LIN {X 0,Y 299.709,Z 498.448,A -85,B 0,C 180,E1 -16464.615,E2 -16464.615} C_VEL
LIN {X 0,Y 299.42,Z 499.838,A -85,B 0,C 180,E1 -16465.959,E2 -16465.959} C_VEL
LIN {X 0,Y 299.059,Z 501.418,A -85,B 0,C 180,E1 -16468.65,E2 -16468.65} C_VEL
LIN {X 0,Y 299.021,Z 501.647,A -85,B 0,C 180,E1 -16469.997,E2 -16469.997} C_VEL
LIN {X 0,Y 299.142,Z 500.888,A -85,B 0,C 180,E1 -16472.69,E2 -16472.69} C_VEL
LIN {X 0,Y 299.43,Z 499.927,A -85,B 0,C 180,E1 -16474.034,E2 -16474.034} C_VEL
LIN {X 0,Y 299.719,Z 498.589,A -85,B 0,C 180,E1 -16475.379,E2 -16475.379} C_VEL
LIN {X 0,Y 300.052,Z 495.813,A -85,B 0,C 180,E1 -16477.398,E2 -16477.398} C_VEL
LIN {X 0,Y 300.857,Z 491.982,A -85,B 0,C 180,E1 -16479.408,E2 -16479.408} C_VEL
LIN {X 0,Y 301.953,Z 486.999,A -85,B 0,C 180,E1 -16481.407,E2 -16481.407} C_VEL
LIN {X 0,Y 302.947,Z 480.761,A -85,B 0,C 180,E1 -16483.41,E2 -16483.41} C_VEL
LIN {X 0,Y 304.253,Z 472.973,A -85,B 0,C 180,E1 -16485.401,E2 -16485.401} C_VEL
LIN {X 0,Y 305.577,Z 464.983,A -85,B 0,C 180,E1 -16487.048,E2 -16487.048} C_VEL
LIN {X 0,Y 306.784,Z 456.263,A -85,B 0,C 180,E1 -16488.53,E2 -16488.53} C_VEL
LIN {X 0,Y 308.051,Z 445.435,A -85,B 0,C 180,E1 -16490.008,E2 -16490.008} C_VEL
LIN {X 0,Y 309.182,Z 435.113,A -85,B 0,C 180,E1 -16491.12,E2 -16491.12} C_VEL
LIN {X 0,Y 310.123,Z 422.899,A -85,B 0,C 180,E1 -16492.151,E2 -16492.151} C_VEL
LIN {X 0,Y 310.297,Z 416.875,A -85,B 0,C 180,E1 -16492.566,E2 -16492.566} C_VEL
LIN {X 0,Y 306.642,Z 404.751,A -85,B 0,C 180,E1 -16493.54,E2 -16493.54} C_VEL
LIN {X 0,Y 303.036,Z 394.815,A -85,B 0,C 180,E1 -16494.215,E2 -16494.215} C_VEL
LIN {X 0,Y 302.843,Z 385.653,A -85,B 0,C 180,E1 -16498.132,E2 -16498.132} C_VEL
LIN {X 0,Y 302.969,Z 376.735,A -85,B 0,C 180,E1 -16502.24,E2 -16502.24} C_VEL
LIN {X 0,Y 303.189,Z 369.244,A -85,B 0,C 180,E1 -16505.775,E2 -16505.775} C_VEL
LIN {X 0,Y 302.932,Z 365.032,A -85,B 0,C 180,E1 -16507.926,E2 -16507.926} C_VEL
LIN {X 0,Y 302.353,Z 361.246,A -85,B 0,C 180,E1 -16509.908,E2 -16509.908} C_VEL
LIN {X 0,Y 300.884,Z 354.027,A -85,B 0,C 180,E1 -16513.606,E2 -16513.606} C_VEL
LIN {X 0,Y 299.828,Z 349.15,A -85,B 0,C 180,E1 -16516.181,E2 -16516.181} C_VEL
LIN {X 0,Y 298.428,Z 343.625,A -85,B 0,C 180,E1 -16519.009,E2 -16519.009} C_VEL
LIN {X 0,Y 298.455,Z 343.623,A -85,B 0,C 180,E1 -16523.183,E2 -16523.183} C_VEL
LIN {X 0,Y 298.378,Z 343.625,A -85,B 0,C 180,E1 -16527.197,E2 -16527.197} C_VEL
LIN {X 0,Y 298.413,Z 343.62,A -85,B 0,C 180,E1 -16530.612,E2 -16530.612} C_VEL
LIN {X 0,Y 298.457,Z 343.611,A -85,B 0,C 180,E1 -16533.659,E2 -16533.659} C_VEL
LIN {X 0,Y 298.458,Z 343.612,A -85,B 0,C 180,E1 -16537.866,E2 -16537.866} C_VEL
LIN {X 0,Y 298.474,Z 343.618,A -85,B 0,C 180,E1 -16539.518,E2 -16539.518} C_VEL
LIN {X 0,Y 297.856,Z 343.69,A -85,B 0,C 180,E1 -16540.645,E2 -16540.645} C_VEL
LIN {X 0,Y 295.029,Z 344.044,A -85,B 0,C 180,E1 -16542.48,E2 -16542.48} C_VEL
LIN {X 0,Y 292.605,Z 344.349,A -85,B 0,C 180,E1 -16543.969,E2 -16543.969} C_VEL
LIN {X 0,Y 291.568,Z 344.467,A -85,B 0,C 180,E1 -16545.122,E2 -16545.122} C_VEL
LIN {X 0,Y 291.487,Z 344.474,A -85,B 0,C 180,E1 -16545.513,E2 -16545.513} C_VEL
LIN {X 0,Y 291.517,Z 344.482,A -85,B 0,C 180,E1 -16548.879,E2 -16548.879} C_VEL
LIN {X 0,Y 291.686,Z 344.456,A -85,B 0,C 180,E1 -16551.687,E2 -16551.687} C_VEL
LIN {X 0,Y 291.607,Z 344.465,A -85,B 0,C 180,E1 -16554.467,E2 -16554.467} C_VEL
LIN {X 0,Y 291.865,Z 344.442,A -85,B 0,C 180,E1 -16558.62,E2 -16558.62} C_VEL
LIN {X 0,Y 291.873,Z 344.427,A -85,B 0,C 180,E1 -16561.379,E2 -16561.379} C_VEL
LIN {X 0,Y 291.615,Z 344.473,A -85,B 0,C 180,E1 -16565.531,E2 -16565.531} C_VEL
LIN {X 0,Y 291.686,Z 344.464,A -85,B 0,C 180,E1 -16568.312,E2 -16568.312} C_VEL
LIN {X 0,Y 291.499,Z 344.489,A -85,B 0,C 180,E1 -16572.532,E2 -16572.532} C_VEL
LIN {X 0,Y 291.533,Z 344.484,A -85,B 0,C 180,E1 -16575.377,E2 -16575.377} C_VEL
LIN {X 0,Y 291.474,Z 344.489,A -85,B 0,C 180,E1 -16579.901,E2 -16579.901} C_VEL
LIN {X 0,Y 291.429,Z 344.53,A -85,B 0,C 180,E1 -16583.728,E2 -16583.728} C_VEL
LIN {X 0,Y 293.265,Z 351.385,A -85,B 0,C 180,E1 -16587.549,E2 -16587.549} C_VEL
LIN {X 0,Y 295.335,Z 359.255,A -85,B 0,C 180,E1 -16591.569,E2 -16591.569} C_VEL
LIN {X 0,Y 297.641,Z 367.228,A -85,B 0,C 180,E1 -16595.345,E2 -16595.345} C_VEL
LIN {X 0,Y 300.221,Z 376.648,A -85,B 0,C 180,E1 -16599.427,E2 -16599.427} C_VEL
LIN {X 0,Y 303.124,Z 387.143,A -85,B 0,C 180,E1 -16603.61,E2 -16603.61} C_VEL
LIN {X 0,Y 305.461,Z 395.462,A -85,B 0,C 180,E1 -16606.692,E2 -16606.692} C_VEL
LIN {X 0,Y 307.2,Z 402.134,A -85,B 0,C 180,E1 -16609.021,E2 -16609.021} C_VEL
LIN {X 0,Y 305.65,Z 408.163,A -85,B 0,C 180,E1 -16610.783,E2 -16610.783} C_VEL
LIN {X 0,Y 304.504,Z 412.249,A -85,B 0,C 180,E1 -16611.963,E2 -16611.963} C_VEL
LIN {X 0,Y 307.508,Z 435.324,A -85,B 0,C 180,E1 -16613.174,E2 -16613.174} C_VEL
LIN {X 0,Y 309.617,Z 451.923,A -85,B 0,C 180,E1 -16614.282,E2 -16614.282} C_VEL
LIN {X 0,Y 311.016,Z 467.45,A -85,B 0,C 180,E1 -16615.51,E2 -16615.51} C_VEL
LIN {X 0,Y 311.129,Z 472.166,A -85,B 0,C 180,E1 -16615.916,E2 -16615.916} C_VEL
LIN {X 0,Y 308.742,Z 487.07,A -85,B 0,C 180,E1 -16617.179,E2 -16617.179} C_VEL
LIN {X 0,Y 306.052,Z 501.73,A -85,B 0,C 180,E1 -16618.703,E2 -16618.703} C_VEL
LIN {X 0,Y 303.557,Z 514.784,A -85,B 0,C 180,E1 -16620.343,E2 -16620.343} C_VEL
LIN {X 0,Y 300.978,Z 527.029,A -85,B 0,C 180,E1 -16622.164,E2 -16622.164} C_VEL
LIN {X 0,Y 298.183,Z 540.238,A -85,B 0,C 180,E1 -16624.528,E2 -16624.528} C_VEL
LIN {X 0,Y 295.85,Z 551.36,A -85,B 0,C 180,E1 -16626.927,E2 -16626.927} C_VEL
LIN {X 0,Y 293.97,Z 560.802,A -85,B 0,C 180,E1 -16629.356,E2 -16629.356} C_VEL
LIN {X 0,Y 292.453,Z 569.92,A -85,B 0,C 180,E1 -16632.162,E2 -16632.162} C_VEL
LIN {X 0,Y 291.413,Z 576.815,A -85,B 0,C 180,E1 -16634.724,E2 -16634.724} C_VEL
LIN {X 0,Y 290.746,Z 582.794,A -85,B 0,C 180,E1 -16637.439,E2 -16637.439} C_VEL
LIN {X 0,Y 290.48,Z 587.668,A -85,B 0,C 180,E1 -16640.253,E2 -16640.253} C_VEL
LIN {X 0,Y 290.473,Z 591.326,A -85,B 0,C 180,E1 -16643.055,E2 -16643.055} C_VEL
LIN {X 0,Y 290.612,Z 593.786,A -85,B 0,C 180,E1 -16645.843,E2 -16645.843} C_VEL
LIN {X 0,Y 290.605,Z 595.006,A -85,B 0,C 180,E1 -16648.618,E2 -16648.618} C_VEL
LIN {X 0,Y 290.576,Z 595.145,A -85,B 0,C 180,E1 -16651.389,E2 -16651.389} C_VEL
LIN {X 0,Y 290.623,Z 594.104,A -85,B 0,C 180,E1 -16654.164,E2 -16654.164} C_VEL
LIN {X 0,Y 290.408,Z 591.736,A -85,B 0,C 180,E1 -16657.158,E2 -16657.158} C_VEL
LIN {X 0,Y 290.35,Z 588.681,A -85,B 0,C 180,E1 -16659.758,E2 -16659.758} C_VEL
LIN {X 0,Y 290.64,Z 584.298,A -85,B 0,C 180,E1 -16662.573,E2 -16662.573} C_VEL
LIN {X 0,Y 291.33,Z 578.847,A -85,B 0,C 180,E1 -16665.392,E2 -16665.392} C_VEL
LIN {X 0,Y 292.839,Z 570.307,A -85,B 0,C 180,E1 -16668.908,E2 -16668.908} C_VEL
LIN {X 0,Y 295.012,Z 560.871,A -85,B 0,C 180,E1 -16672.066,E2 -16672.066} C_VEL
LIN {X 0,Y 297.929,Z 549.828,A -85,B 0,C 180,E1 -16675.129,E2 -16675.129} C_VEL
LIN {X 0,Y 301.401,Z 538.282,A -85,B 0,C 180,E1 -16677.801,E2 -16677.801} C_VEL
LIN {X 0,Y 305.467,Z 524.903,A -85,B 0,C 180,E1 -16680.412,E2 -16680.412} C_VEL
LIN {X 0,Y 310.085,Z 510.339,A -85,B 0,C 180,E1 -16682.763,E2 -16682.763} C_VEL
LIN {X 0,Y 314.614,Z 495.802,A -85,B 0,C 180,E1 -16684.727,E2 -16684.727} C_VEL
LIN {X 0,Y 319.648,Z 479.136,A -85,B 0,C 180,E1 -16686.567,E2 -16686.567} C_VEL
LIN {X 0,Y 320.589,Z 474.856,A -85,B 0,C 180,E1 -16687.038,E2 -16687.038} C_VEL
LIN {X 0,Y 322.54,Z 461.569,A -85,B 0,C 180,E1 -16688.591,E2 -16688.591} C_VEL
LIN {X 0,Y 323.882,Z 451.061,A -85,B 0,C 180,E1 -16689.761,E2 -16689.761} C_VEL
LIN {X 0,Y 324.459,Z 439.447,A -85,B 0,C 180,E1 -16691.255,E2 -16691.255} C_VEL
LIN {X 0,Y 324.455,Z 428.956,A -85,B 0,C 180,E1 -16692.817,E2 -16692.817} C_VEL
LIN {X 0,Y 324.347,Z 427.026,A -85,B 0,C 180,E1 -16693.153,E2 -16693.153} C_VEL
LIN {X 0,Y 323.2,Z 424.156,A -85,B 0,C 180,E1 -16694.145,E2 -16694.145} C_VEL
LIN {X 0,Y 321.573,Z 421.326,A -85,B 0,C 180,E1 -16695.625,E2 -16695.625} C_VEL
LIN {X 0,Y 320.315,Z 419.287,A -85,B 0,C 180,E1 -16697.144,E2 -16697.144} C_VEL
LIN {X 0,Y 319.502,Z 417.856,A -85,B 0,C 180,E1 -16698.708,E2 -16698.708} C_VEL
LIN {X 0,Y 319.091,Z 417.219,A -85,B 0,C 180,E1 -16700.436,E2 -16700.436} C_VEL
LIN {X 0,Y 319.182,Z 417.312,A -85,B 0,C 180,E1 -16701.938,E2 -16701.938} C_VEL
LIN {X 0,Y 319.666,Z 420.051,A -85,B 0,C 180,E1 -16704.439,E2 -16704.439} C_VEL
LIN {X 0,Y 320.351,Z 423.999,A -85,B 0,C 180,E1 -16706.48,E2 -16706.48} C_VEL
LIN {X 0,Y 321.491,Z 428.847,A -85,B 0,C 180,E1 -16708.496,E2 -16708.496} C_VEL
LIN {X 0,Y 322.7,Z 435.191,A -85,B 0,C 180,E1 -16710.596,E2 -16710.596} C_VEL
LIN {X 0,Y 323.498,Z 442.422,A -85,B 0,C 180,E1 -16712.558,E2 -16712.558} C_VEL
LIN {X 0,Y 322.358,Z 446.313,A -85,B 0,C 180,E1 -16713.104,E2 -16713.104} C_VEL
LIN {X 0,Y 318.092,Z 458.146,A -85,B 0,C 180,E1 -16714.83,E2 -16714.83} C_VEL
LIN {X 0,Y 313.751,Z 469.712,A -85,B 0,C 180,E1 -16716.922,E2 -16716.922} C_VEL
LIN {X 0,Y 310.415,Z 478.194,A -85,B 0,C 180,E1 -16718.762,E2 -16718.762} C_VEL
LIN {X 0,Y 306.945,Z 486.567,A -85,B 0,C 180,E1 -16720.958,E2 -16720.958} C_VEL
LIN {X 0,Y 303.836,Z 493.445,A -85,B 0,C 180,E1 -16723.194,E2 -16723.194} C_VEL
LIN {X 0,Y 300.755,Z 499.656,A -85,B 0,C 180,E1 -16725.797,E2 -16725.797} C_VEL
LIN {X 0,Y 298.775,Z 503.283,A -85,B 0,C 180,E1 -16727.778,E2 -16727.778} C_VEL
LIN {X 0,Y 296.676,Z 506.657,A -85,B 0,C 180,E1 -16730.455,E2 -16730.455} C_VEL
LIN {X 0,Y 295.821,Z 507.785,A -85,B 0,C 180,E1 -16731.805,E2 -16731.805} C_VEL
LIN {X 0,Y 295.166,Z 508.504,A -85,B 0,C 180,E1 -16733.163,E2 -16733.163} C_VEL
LIN {X 0,Y 293.913,Z 508.817,A -85,B 0,C 180,E1 -16735.887,E2 -16735.887} C_VEL
LIN {X 0,Y 293.36,Z 508.405,A -85,B 0,C 180,E1 -16737.254,E2 -16737.254} C_VEL
LIN {X 0,Y 292.952,Z 507.587,A -85,B 0,C 180,E1 -16738.626,E2 -16738.626} C_VEL
LIN {X 0,Y 292.613,Z 506.375,A -85,B 0,C 180,E1 -16740.001,E2 -16740.001} C_VEL
LIN {X 0,Y 292.392,Z 503.757,A -85,B 0,C 180,E1 -16742.067,E2 -16742.067} C_VEL
LIN {X 0,Y 292.397,Z 500.192,A -85,B 0,C 180,E1 -16744.136,E2 -16744.136} C_VEL
LIN {X 0,Y 292.337,Z 495.653,A -85,B 0,C 180,E1 -16746.211,E2 -16746.211} C_VEL
LIN {X 0,Y 292.947,Z 488.932,A -85,B 0,C 180,E1 -16748.624,E2 -16748.624} C_VEL
LIN {X 0,Y 293.557,Z 480.592,A -85,B 0,C 180,E1 -16751.042,E2 -16751.042} C_VEL
LIN {X 0,Y 294.384,Z 471.876,A -85,B 0,C 180,E1 -16753.109,E2 -16753.109} C_VEL
LIN {X 0,Y 295.367,Z 461.466,A -85,B 0,C 180,E1 -16755.174,E2 -16755.174} C_VEL
LIN {X 0,Y 296.644,Z 450.12,A -85,B 0,C 180,E1 -16757.049,E2 -16757.049} C_VEL
LIN {X 0,Y 297.862,Z 437.703,A -85,B 0,C 180,E1 -16758.753,E2 -16758.753} C_VEL
LIN {X 0,Y 299.01,Z 424.062,A -85,B 0,C 180,E1 -16760.305,E2 -16760.305} C_VEL
LIN {X 0,Y 300.202,Z 410.631,A -85,B 0,C 180,E1 -16761.547,E2 -16761.547} C_VEL
LIN {X 0,Y 296.859,Z 394.61,A -85,B 0,C 180,E1 -16763.018,E2 -16763.018} C_VEL
LIN {X 0,Y 293.024,Z 378.623,A -85,B 0,C 180,E1 -16764.237,E2 -16764.237} C_VEL
LIN {X 0,Y 292.023,Z 374.499,A -85,B 0,C 180,E1 -16764.54,E2 -16764.54} C_VEL
LIN {X 0,Y 292.382,Z 369.177,A -85,B 0,C 180,E1 -16767.952,E2 -16767.952} C_VEL
LIN {X 0,Y 292.834,Z 363.258,A -85,B 0,C 180,E1 -16771.871,E2 -16771.871} C_VEL
LIN {X 0,Y 293.207,Z 358.041,A -85,B 0,C 180,E1 -16775.413,E2 -16775.413} C_VEL
LIN {X 0,Y 292.974,Z 353.615,A -85,B 0,C 180,E1 -16778.588,E2 -16778.588} C_VEL
LIN {X 0,Y 292.196,Z 348.783,A -85,B 0,C 180,E1 -16782.336,E2 -16782.336} C_VEL
LIN {X 0,Y 293.162,Z 351.814,A -85,B 0,C 180,E1 -16784.045,E2 -16784.045} C_VEL
LIN {X 0,Y 294.906,Z 359.618,A -85,B 0,C 180,E1 -16788.139,E2 -16788.139} C_VEL
LIN {X 0,Y 296.129,Z 366.652,A -85,B 0,C 180,E1 -16791.895,E2 -16791.895} C_VEL
LIN {X 0,Y 296.461,Z 370.31,A -85,B 0,C 180,E1 -16793.709,E2 -16793.709} C_VEL
LIN {X 0,Y 296.218,Z 378.746,A -85,B 0,C 180,E1 -16797.732,E2 -16797.732} C_VEL
LIN {X 0,Y 296.115,Z 389.045,A -85,B 0,C 180,E1 -16802.428,E2 -16802.428} C_VEL
LIN {X 0,Y 296.28,Z 395.804,A -85,B 0,C 180,E1 -16805.308,E2 -16805.308} C_VEL
LIN {X 0,Y 301.098,Z 409.41,A -85,B 0,C 180,E1 -16806.291,E2 -16806.291} C_VEL
LIN {X 0,Y 303.862,Z 419.007,A -85,B 0,C 180,E1 -16807.118,E2 -16807.118} C_VEL
LIN {X 0,Y 302.971,Z 431.867,A -85,B 0,C 180,E1 -16808.108,E2 -16808.108} C_VEL
LIN {X 0,Y 301.875,Z 443.495,A -85,B 0,C 180,E1 -16809.292,E2 -16809.292} C_VEL
LIN {X 0,Y 300.567,Z 454.315,A -85,B 0,C 180,E1 -16810.711,E2 -16810.711} C_VEL
LIN {X 0,Y 299.179,Z 463.594,A -85,B 0,C 180,E1 -16812.216,E2 -16812.216} C_VEL
LIN {X 0,Y 297.83,Z 472.044,A -85,B 0,C 180,E1 -16813.9,E2 -16813.9} C_VEL
LIN {X 0,Y 296.362,Z 480.26,A -85,B 0,C 180,E1 -16815.929,E2 -16815.929} C_VEL
LIN {X 0,Y 295.496,Z 485.81,A -85,B 0,C 180,E1 -16817.637,E2 -16817.637} C_VEL
LIN {X 0,Y 294.347,Z 491.24,A -85,B 0,C 180,E1 -16819.681,E2 -16819.681} C_VEL
LIN {X 0,Y 293.252,Z 495.521,A -85,B 0,C 180,E1 -16821.729,E2 -16821.729} C_VEL
LIN {X 0,Y 292.874,Z 497.74,A -85,B 0,C 180,E1 -16823.106,E2 -16823.106} C_VEL
LIN {X 0,Y 292.725,Z 499.525,A -85,B 0,C 180,E1 -16824.486,E2 -16824.486} C_VEL
LIN {X 0,Y 292.421,Z 500.915,A -85,B 0,C 180,E1 -16825.862,E2 -16825.862} C_VEL
LIN {X 0,Y 292.053,Z 502.493,A -85,B 0,C 180,E1 -16828.618,E2 -16828.618} C_VEL
LIN {X 0,Y 292.01,Z 502.723,A -85,B 0,C 180,E1 -16829.997,E2 -16829.997} C_VEL
LIN {X 0,Y 292.132,Z 501.964,A -85,B 0,C 180,E1 -16832.754,E2 -16832.754} C_VEL
LIN {X 0,Y 292.431,Z 501.003,A -85,B 0,C 180,E1 -16834.131,E2 -16834.131} C_VEL
LIN {X 0,Y 292.732,Z 499.664,A -85,B 0,C 180,E1 -16835.507,E2 -16835.507} C_VEL
LIN {X 0,Y 293.091,Z 496.889,A -85,B 0,C 180,E1 -16837.575,E2 -16837.575} C_VEL
LIN {X 0,Y 293.935,Z 493.056,A -85,B 0,C 180,E1 -16839.631,E2 -16839.631} C_VEL
LIN {X 0,Y 295.08,Z 488.072,A -85,B 0,C 180,E1 -16841.676,E2 -16841.676} C_VEL
LIN {X 0,Y 296.126,Z 481.832,A -85,B 0,C 180,E1 -16843.725,E2 -16843.725} C_VEL
LIN {X 0,Y 297.504,Z 474.04,A -85,B 0,C 180,E1 -16845.76,E2 -16845.76} C_VEL
LIN {X 0,Y 298.872,Z 466.05,A -85,B 0,C 180,E1 -16847.443,E2 -16847.443} C_VEL
LIN {X 0,Y 300.297,Z 456.215,A -85,B 0,C 180,E1 -16849.122,E2 -16849.122} C_VEL
LIN {X 0,Y 301.463,Z 446.492,A -85,B 0,C 180,E1 -16850.465,E2 -16850.465} C_VEL
LIN {X 0,Y 302.661,Z 436.146,A -85,B 0,C 180,E1 -16851.599,E2 -16851.599} C_VEL
LIN {X 0,Y 303.614,Z 424.465,A -85,B 0,C 180,E1 -16852.608,E2 -16852.608} C_VEL
LIN {X 0,Y 303.848,Z 418.707,A -85,B 0,C 180,E1 -16853.019,E2 -16853.019} C_VEL
LIN {X 0,Y 300.261,Z 406.801,A -85,B 0,C 180,E1 -16854.025,E2 -16854.025} C_VEL
LIN {X 0,Y 296.28,Z 395.811,A -85,B 0,C 180,E1 -16854.818,E2 -16854.818} C_VEL
LIN {X 0,Y 296.092,Z 387.112,A -85,B 0,C 180,E1 -16858.57,E2 -16858.57} C_VEL
LIN {X 0,Y 296.229,Z 379.14,A -85,B 0,C 180,E1 -16862.259,E2 -16862.259} C_VEL
LIN {X 0,Y 296.485,Z 370.58,A -85,B 0,C 180,E1 -16866.337,E2 -16866.337} C_VEL
LIN {X 0,Y 296.007,Z 365.472,A -85,B 0,C 180,E1 -16869.035,E2 -16869.035} C_VEL
LIN {X 0,Y 294.773,Z 359.052,A -85,B 0,C 180,E1 -16872.344,E2 -16872.344} C_VEL
LIN {X 0,Y 293.345,Z 352.213,A -85,B 0,C 180,E1 -16875.989,E2 -16875.989} C_VEL
LIN {X 0,Y 291.502,Z 345.062,A -85,B 0,C 180,E1 -16879.703,E2 -16879.703} C_VEL
LIN {X 0,Y 291.398,Z 344.498,A -85,B 0,C 180,E1 -16880.001,E2 -16880.001} C_VEL
LIN {X 0,Y 291.418,Z 344.499,A -85,B 0,C 180,E1 -16882.92,E2 -16882.92} C_VEL
LIN {X 0,Y 291.328,Z 344.506,A -85,B 0,C 180,E1 -16886.299,E2 -16886.299} C_VEL
LIN {X 0,Y 291.369,Z 344.496,A -85,B 0,C 180,E1 -16890.258,E2 -16890.258} C_VEL
LIN {X 0,Y 291.405,Z 344.492,A -85,B 0,C 180,E1 -16894.27,E2 -16894.27} C_VEL
LIN {X 0,Y 291.414,Z 344.487,A -85,B 0,C 180,E1 -16897.302,E2 -16897.302} C_VEL
LIN {X 0,Y 291.493,Z 344.483,A -85,B 0,C 180,E1 -16900.272,E2 -16900.272} C_VEL
LIN {X 0,Y 291.519,Z 344.477,A -85,B 0,C 180,E1 -16904.633,E2 -16904.633} C_VEL
LIN {X 0,Y 291.487,Z 344.474,A -85,B 0,C 180,E1 -16905.513,E2 -16905.513} C_VEL
LIN {X 0,Y 290.85,Z 344.559,A -85,B 0,C 180,E1 -16906.666,E2 -16906.666} C_VEL
LIN {X 0,Y 288.088,Z 344.912,A -85,B 0,C 180,E1 -16908.546,E2 -16908.546} C_VEL
LIN {X 0,Y 285.734,Z 345.2,A -85,B 0,C 180,E1 -16910.071,E2 -16910.071} C_VEL
LIN {X 0,Y 284.718,Z 345.322,A -85,B 0,C 180,E1 -16911.251,E2 -16911.251} C_VEL
LIN {X 0,Y 284.632,Z 345.333,A -85,B 0,C 180,E1 -16911.651,E2 -16911.651} C_VEL
LIN {X 0,Y 284.578,Z 345.342,A -85,B 0,C 180,E1 -16914.33,E2 -16914.33} C_VEL
LIN {X 0,Y 284.832,Z 345.318,A -85,B 0,C 180,E1 -16918.586,E2 -16918.586} C_VEL
LIN {X 0,Y 284.839,Z 345.303,A -85,B 0,C 180,E1 -16921.413,E2 -16921.413} C_VEL
LIN {X 0,Y 284.585,Z 345.35,A -85,B 0,C 180,E1 -16925.669,E2 -16925.669} C_VEL
LIN {X 0,Y 284.643,Z 345.341,A -85,B 0,C 180,E1 -16929.054,E2 -16929.054} C_VEL
LIN {X 0,Y 284.455,Z 345.365,A -85,B 0,C 180,E1 -16932.847,E2 -16932.847} C_VEL
LIN {X 0,Y 284.466,Z 345.365,A -85,B 0,C 180,E1 -16935.769,E2 -16935.769} C_VEL
LIN {X 0,Y 284.406,Z 345.369,A -85,B 0,C 180,E1 -16940.24,E2 -16940.24} C_VEL
LIN {X 0,Y 284.407,Z 345.509,A -85,B 0,C 180,E1 -16942.616,E2 -16942.616} C_VEL
LIN {X 0,Y 286.043,Z 351.774,A -85,B 0,C 180,E1 -16946.247,E2 -16946.247} C_VEL
LIN {X 0,Y 287.963,Z 358.811,A -85,B 0,C 180,E1 -16950.021,E2 -16950.021} C_VEL
LIN {X 0,Y 290.093,Z 366.587,A -85,B 0,C 180,E1 -16953.863,E2 -16953.863} C_VEL
LIN {X 0,Y 292.27,Z 374.529,A -85,B 0,C 180,E1 -16957.491,E2 -16957.491} C_VEL
LIN {X 0,Y 294.552,Z 382.807,A -85,B 0,C 180,E1 -16961.006,E2 -16961.006} C_VEL
LIN {X 0,Y 297.528,Z 393.255,A -85,B 0,C 180,E1 -16965.124,E2 -16965.124} C_VEL
LIN {X 0,Y 300.006,Z 402.705,A -85,B 0,C 180,E1 -16968.558,E2 -16968.558} C_VEL
LIN {X 0,Y 300.174,Z 404.143,A -85,B 0,C 180,E1 -16969.043,E2 -16969.043} C_VEL
LIN {X 0,Y 297.875,Z 412.008,A -85,B 0,C 180,E1 -16971.379,E2 -16971.379} C_VEL
LIN {X 0,Y 300.73,Z 434.611,A -85,B 0,C 180,E1 -16972.57,E2 -16972.57} C_VEL
LIN {X 0,Y 302.52,Z 449.258,A -85,B 0,C 180,E1 -16973.548,E2 -16973.548} C_VEL
LIN {X 0,Y 304.076,Z 465.037,A -85,B 0,C 180,E1 -16974.816,E2 -16974.816} C_VEL
LIN {X 0,Y 304.479,Z 472.307,A -85,B 0,C 180,E1 -16975.467,E2 -16975.467} C_VEL
LIN {X 0,Y 301.82,Z 488.204,A -85,B 0,C 180,E1 -16976.868,E2 -16976.868} C_VEL
LIN {X 0,Y 299.001,Z 502.917,A -85,B 0,C 180,E1 -16978.472,E2 -16978.472} C_VEL
LIN {X 0,Y 296.435,Z 515.616,A -85,B 0,C 180,E1 -16980.145,E2 -16980.145} C_VEL
LIN {X 0,Y 293.704,Z 528.288,A -85,B 0,C 180,E1 -16982.128,E2 -16982.128} C_VEL
LIN {X 0,Y 291.234,Z 539.758,A -85,B 0,C 180,E1 -16984.259,E2 -16984.259} C_VEL
LIN {X 0,Y 288.848,Z 550.829,A -85,B 0,C 180,E1 -16986.715,E2 -16986.715} C_VEL
LIN {X 0,Y 286.954,Z 560.211,A -85,B 0,C 180,E1 -16989.203,E2 -16989.203} C_VEL
LIN {X 0,Y 285.395,Z 569.257,A -85,B 0,C 180,E1 -16992.076,E2 -16992.076} C_VEL
LIN {X 0,Y 284.231,Z 576.989,A -85,B 0,C 180,E1 -16995.096,E2 -16995.096} C_VEL
LIN {X 0,Y 283.672,Z 582.686,A -85,B 0,C 180,E1 -16997.847,E2 -16997.847} C_VEL
LIN {X 0,Y 283.434,Z 587.361,A -85,B 0,C 180,E1 -17000.729,E2 -17000.729} C_VEL
LIN {X 0,Y 283.479,Z 590.049,A -85,B 0,C 180,E1 -17002.883,E2 -17002.883} C_VEL
LIN {X 0,Y 283.587,Z 592.542,A -85,B 0,C 180,E1 -17005.74,E2 -17005.74} C_VEL
LIN {X 0,Y 283.596,Z 593.839,A -85,B 0,C 180,E1 -17008.583,E2 -17008.583} C_VEL
LIN {X 0,Y 283.56,Z 594.03,A -85,B 0,C 180,E1 -17011.424,E2 -17011.424} C_VEL
LIN {X 0,Y 283.591,Z 593.024,A -85,B 0,C 180,E1 -17014.267,E2 -17014.267} C_VEL
LIN {X 0,Y 283.351,Z 590.857,A -85,B 0,C 180,E1 -17017.2,E2 -17017.2} C_VEL
LIN {X 0,Y 283.28,Z 587.686,A -85,B 0,C 180,E1 -17020.004,E2 -17020.004} C_VEL
LIN {X 0,Y 283.603,Z 583.386,A -85,B 0,C 180,E1 -17022.89,E2 -17022.89} C_VEL
LIN {X 0,Y 284.342,Z 577.983,A -85,B 0,C 180,E1 -17025.78,E2 -17025.78} C_VEL
LIN {X 0,Y 285.569,Z 571.386,A -85,B 0,C 180,E1 -17028.662,E2 -17028.662} C_VEL
LIN {X 0,Y 287.581,Z 562.85,A -85,B 0,C 180,E1 -17031.775,E2 -17031.775} C_VEL
LIN {X 0,Y 290.234,Z 553.302,A -85,B 0,C 180,E1 -17034.693,E2 -17034.693} C_VEL
LIN {X 0,Y 293.823,Z 541.818,A -85,B 0,C 180,E1 -17037.629,E2 -17037.629} C_VEL
LIN {X 0,Y 297.617,Z 530.286,A -85,B 0,C 180,E1 -17040.122,E2 -17040.122} C_VEL
LIN {X 0,Y 302.489,Z 516.005,A -85,B 0,C 180,E1 -17042.699,E2 -17042.699} C_VEL
LIN {X 0,Y 307.398,Z 501.59,A -85,B 0,C 180,E1 -17044.863,E2 -17044.863} C_VEL
LIN {X 0,Y 312.17,Z 487.424,A -85,B 0,C 180,E1 -17046.63,E2 -17046.63} C_VEL
LIN {X 0,Y 315.197,Z 477.495,A -85,B 0,C 180,E1 -17047.725,E2 -17047.725} C_VEL
LIN {X 0,Y 317.501,Z 464.627,A -85,B 0,C 180,E1 -17049.327,E2 -17049.327} C_VEL
LIN {X 0,Y 319.351,Z 453.739,A -85,B 0,C 180,E1 -17050.607,E2 -17050.607} C_VEL
LIN {X 0,Y 320.344,Z 442.456,A -85,B 0,C 180,E1 -17052.137,E2 -17052.137} C_VEL
LIN {X 0,Y 320.788,Z 432.6,A -85,B 0,C 180,E1 -17053.699,E2 -17053.699} C_VEL
LIN {X 0,Y 319.912,Z 429.825,A -85,B 0,C 180,E1 -17054.671,E2 -17054.671} C_VEL
LIN {X 0,Y 317.988,Z 426.453,A -85,B 0,C 180,E1 -17056.754,E2 -17056.754} C_VEL
LIN {X 0,Y 316.786,Z 424.341,A -85,B 0,C 180,E1 -17058.968,E2 -17058.968} C_VEL
LIN {X 0,Y 316.365,Z 423.813,A -85,B 0,C 180,E1 -17061.537,E2 -17061.537} C_VEL
LIN {X 0,Y 316.5,Z 426.109,A -85,B 0,C 180,E1 -17064.028,E2 -17064.028} C_VEL
LIN {X 0,Y 316.78,Z 428.779,A -85,B 0,C 180,E1 -17065.626,E2 -17065.626} C_VEL
LIN {X 0,Y 317.486,Z 433.861,A -85,B 0,C 180,E1 -17067.909,E2 -17067.909} C_VEL
LIN {X 0,Y 318.083,Z 438.239,A -85,B 0,C 180,E1 -17069.512,E2 -17069.512} C_VEL
LIN {X 0,Y 318.614,Z 444.125,A -85,B 0,C 180,E1 -17071.326,E2 -17071.326} C_VEL
LIN {X 0,Y 318.599,Z 446.482,A -85,B 0,C 180,E1 -17071.933,E2 -17071.933} C_VEL
LIN {X 0,Y 313.832,Z 458.914,A -85,B 0,C 180,E1 -17073.751,E2 -17073.751} C_VEL
LIN {X 0,Y 309.106,Z 470.425,A -85,B 0,C 180,E1 -17075.842,E2 -17075.842} C_VEL
LIN {X 0,Y 305.061,Z 479.771,A -85,B 0,C 180,E1 -17077.914,E2 -17077.914} C_VEL
LIN {X 0,Y 301.2,Z 488.323,A -85,B 0,C 180,E1 -17080.225,E2 -17080.225} C_VEL
LIN {X 0,Y 298.329,Z 494.204,A -85,B 0,C 180,E1 -17082.167,E2 -17082.167} C_VEL
LIN {X 0,Y 295.005,Z 500.52,A -85,B 0,C 180,E1 -17084.808,E2 -17084.808} C_VEL
LIN {X 0,Y 292.115,Z 505.237,A -85,B 0,C 180,E1 -17087.495,E2 -17087.495} C_VEL
LIN {X 0,Y 289.908,Z 508.421,A -85,B 0,C 180,E1 -17090.23,E2 -17090.23} C_VEL
LIN {X 0,Y 288.287,Z 510.026,A -85,B 0,C 180,E1 -17092.999,E2 -17092.999} C_VEL
LIN {X 0,Y 286.961,Z 510.141,A -85,B 0,C 180,E1 -17095.787,E2 -17095.787} C_VEL
LIN {X 0,Y 285.951,Z 508.743,A -85,B 0,C 180,E1 -17098.592,E2 -17098.592} C_VEL
LIN {X 0,Y 285.599,Z 507.45,A -85,B 0,C 180,E1 -17100.001,E2 -17100.001} C_VEL
LIN {X 0,Y 285.36,Z 504.691,A -85,B 0,C 180,E1 -17102.118,E2 -17102.118} C_VEL
LIN {X 0,Y 285.382,Z 500.98,A -85,B 0,C 180,E1 -17104.237,E2 -17104.237} C_VEL
LIN {X 0,Y 285.323,Z 496.3,A -85,B 0,C 180,E1 -17106.364,E2 -17106.364} C_VEL
LIN {X 0,Y 285.961,Z 489.426,A -85,B 0,C 180,E1 -17108.836,E2 -17108.836} C_VEL
LIN {X 0,Y 286.6,Z 480.915,A -85,B 0,C 180,E1 -17111.314,E2 -17111.314} C_VEL
LIN {X 0,Y 287.438,Z 472.012,A -85,B 0,C 180,E1 -17113.432,E2 -17113.432} C_VEL
LIN {X 0,Y 288.465,Z 461.403,A -85,B 0,C 180,E1 -17115.546,E2 -17115.546} C_VEL
LIN {X 0,Y 289.825,Z 449.814,A -85,B 0,C 180,E1 -17117.463,E2 -17117.463} C_VEL
LIN {X 0,Y 291.216,Z 435.81,A -85,B 0,C 180,E1 -17119.381,E2 -17119.381} C_VEL
LIN {X 0,Y 292.448,Z 422.003,A -85,B 0,C 180,E1 -17120.927,E2 -17120.927} C_VEL
LIN {X 0,Y 293.347,Z 411.729,A -85,B 0,C 180,E1 -17121.889,E2 -17121.889} C_VEL
LIN {X 0,Y 290.216,Z 396.576,A -85,B 0,C 180,E1 -17123.325,E2 -17123.325} C_VEL
LIN {X 0,Y 286.689,Z 381.561,A -85,B 0,C 180,E1 -17124.529,E2 -17124.529} C_VEL
LIN {X 0,Y 285.049,Z 374.919,A -85,B 0,C 180,E1 -17125.025,E2 -17125.025} C_VEL
LIN {X 0,Y 285.587,Z 368.101,A -85,B 0,C 180,E1 -17129.485,E2 -17129.485} C_VEL
LIN {X 0,Y 286.011,Z 362.421,A -85,B 0,C 180,E1 -17133.332,E2 -17133.332} C_VEL
LIN {X 0,Y 286.196,Z 358.446,A -85,B 0,C 180,E1 -17136.112,E2 -17136.112} C_VEL
LIN {X 0,Y 285.958,Z 354.675,A -85,B 0,C 180,E1 -17138.873,E2 -17138.873} C_VEL
LIN {X 0,Y 285.335,Z 350.833,A -85,B 0,C 180,E1 -17141.92,E2 -17141.92} C_VEL
LIN {X 0,Y 286.647,Z 354.638,A -85,B 0,C 180,E1 -17144.064,E2 -17144.064} C_VEL
LIN {X 0,Y 288.225,Z 361.926,A -85,B 0,C 180,E1 -17147.981,E2 -17147.981} C_VEL
LIN {X 0,Y 289.266,Z 367.635,A -85,B 0,C 180,E1 -17151.03,E2 -17151.03} C_VEL
LIN {X 0,Y 289.74,Z 371.784,A -85,B 0,C 180,E1 -17153.175,E2 -17153.175} C_VEL
LIN {X 0,Y 289.539,Z 379.493,A -85,B 0,C 180,E1 -17156.894,E2 -17156.894} C_VEL
LIN {X 0,Y 289.363,Z 388.266,A -85,B 0,C 180,E1 -17160.971,E2 -17160.971} C_VEL
LIN {X 0,Y 289.529,Z 396.869,A -85,B 0,C 180,E1 -17164.711,E2 -17164.711} C_VEL
LIN {X 0,Y 294.179,Z 409.674,A -85,B 0,C 180,E1 -17165.652,E2 -17165.652} C_VEL
LIN {X 0,Y 297.311,Z 420.264,A -85,B 0,C 180,E1 -17166.599,E2 -17166.599} C_VEL
LIN {X 0,Y 296.498,Z 432.72,A -85,B 0,C 180,E1 -17167.584,E2 -17167.584} C_VEL
LIN {X 0,Y 295.324,Z 444.516,A -85,B 0,C 180,E1 -17168.805,E2 -17168.805} C_VEL
LIN {X 0,Y 293.95,Z 455.384,A -85,B 0,C 180,E1 -17170.259,E2 -17170.259} C_VEL
LIN {X 0,Y 292.519,Z 464.663,A -85,B 0,C 180,E1 -17171.797,E2 -17171.797} C_VEL
LIN {X 0,Y 291.095,Z 473.118,A -85,B 0,C 180,E1 -17173.517,E2 -17173.517} C_VEL
LIN {X 0,Y 289.561,Z 481.336,A -85,B 0,C 180,E1 -17175.591,E2 -17175.591} C_VEL
LIN {X 0,Y 288.652,Z 486.885,A -85,B 0,C 180,E1 -17177.339,E2 -17177.339} C_VEL
LIN {X 0,Y 287.446,Z 492.316,A -85,B 0,C 180,E1 -17179.43,E2 -17179.43} C_VEL
LIN {X 0,Y 286.31,Z 496.598,A -85,B 0,C 180,E1 -17181.527,E2 -17181.527} C_VEL
LIN {X 0,Y 285.909,Z 498.817,A -85,B 0,C 180,E1 -17182.937,E2 -17182.937} C_VEL
LIN {X 0,Y 285.74,Z 500.602,A -85,B 0,C 180,E1 -17184.351,E2 -17184.351} C_VEL
LIN {X 0,Y 285.422,Z 501.992,A -85,B 0,C 180,E1 -17185.76,E2 -17185.76} C_VEL
LIN {X 0,Y 285.044,Z 503.569,A -85,B 0,C 180,E1 -17188.584,E2 -17188.584} C_VEL
LIN {X 0,Y 285.019,Z 503.796,A -85,B 0,C 180,E1 -17189.997,E2 -17189.997} C_VEL
LIN {X 0,Y 285.124,Z 503.041,A -85,B 0,C 180,E1 -17192.822,E2 -17192.822} C_VEL
LIN {X 0,Y 285.432,Z 502.079,A -85,B 0,C 180,E1 -17194.233,E2 -17194.233} C_VEL
LIN {X 0,Y 285.746,Z 500.741,A -85,B 0,C 180,E1 -17195.642,E2 -17195.642} C_VEL
LIN {X 0,Y 286.133,Z 497.964,A -85,B 0,C 180,E1 -17197.76,E2 -17197.76} C_VEL
LIN {X 0,Y 287.019,Z 494.131,A -85,B 0,C 180,E1 -17199.866,E2 -17199.866} C_VEL
LIN {X 0,Y 288.213,Z 489.145,A -85,B 0,C 180,E1 -17201.959,E2 -17201.959} C_VEL
LIN {X 0,Y 289.312,Z 482.904,A -85,B 0,C 180,E1 -17204.055,E2 -17204.055} C_VEL
LIN {X 0,Y 290.775,Z 475.107,A -85,B 0,C 180,E1 -17206.134,E2 -17206.134} C_VEL
LIN {X 0,Y 292.182,Z 467.116,A -85,B 0,C 180,E1 -17207.855,E2 -17207.855} C_VEL
LIN {X 0,Y 293.678,Z 457.277,A -85,B 0,C 180,E1 -17209.571,E2 -17209.571} C_VEL
LIN {X 0,Y 294.894,Z 447.55,A -85,B 0,C 180,E1 -17210.942,E2 -17210.942} C_VEL
LIN {X 0,Y 296.149,Z 437.135,A -85,B 0,C 180,E1 -17212.106,E2 -17212.106} C_VEL
LIN {X 0,Y 297.113,Z 425.787,A -85,B 0,C 180,E1 -17213.107,E2 -17213.107} C_VEL
LIN {X 0,Y 297.414,Z 421.198,A -85,B 0,C 180,E1 -17213.437,E2 -17213.437} C_VEL
LIN {X 0,Y 294.605,Z 410.997,A -85,B 0,C 180,E1 -17214.351,E2 -17214.351} C_VEL
LIN {X 0,Y 290.422,Z 399.211,A -85,B 0,C 180,E1 -17215.251,E2 -17215.251} C_VEL
LIN {X 0,Y 289.506,Z 396.85,A -85,B 0,C 180,E1 -17215.44,E2 -17215.44} C_VEL
LIN {X 0,Y 289.388,Z 388.515,A -85,B 0,C 180,E1 -17219.055,E2 -17219.055} C_VEL
LIN {X 0,Y 289.571,Z 379.831,A -85,B 0,C 180,E1 -17223.094,E2 -17223.094} C_VEL
LIN {X 0,Y 289.822,Z 373.437,A -85,B 0,C 180,E1 -17226.2,E2 -17226.2} C_VEL
LIN {X 0,Y 289.541,Z 369.543,A -85,B 0,C 180,E1 -17228.154,E2 -17228.154} C_VEL
LIN {X 0,Y 288.637,Z 364.019,A -85,B 0,C 180,E1 -17231.098,E2 -17231.098} C_VEL
LIN {X 0,Y 287.114,Z 356.389,A -85,B 0,C 180,E1 -17235.218,E2 -17235.218} C_VEL
LIN {X 0,Y 285.635,Z 350.337,A -85,B 0,C 180,E1 -17238.368,E2 -17238.368} C_VEL
LIN {X 0,Y 284.328,Z 345.379,A -85,B 0,C 180,E1 -17241.154,E2 -17241.154} C_VEL
LIN {X 0,Y 284.346,Z 345.374,A -85,B 0,C 180,E1 -17244.643,E2 -17244.643} C_VEL
LIN {X 0,Y 284.278,Z 345.389,A -85,B 0,C 180,E1 -17248.723,E2 -17248.723} C_VEL
LIN {X 0,Y 284.379,Z 345.367,A -85,B 0,C 180,E1 -17252.824,E2 -17252.824} C_VEL
LIN {X 0,Y 284.376,Z 345.365,A -85,B 0,C 180,E1 -17256.707,E2 -17256.707} C_VEL
LIN {X 0,Y 284.416,Z 345.367,A -85,B 0,C 180,E1 -17259.869,E2 -17259.869} C_VEL
LIN {X 0,Y 284.457,Z 345.359,A -85,B 0,C 180,E1 -17264.468,E2 -17264.468} C_VEL
LIN {X 0,Y 284.469,Z 345.362,A -85,B 0,C 180,E1 -17268.6,E2 -17268.6} C_VEL
LIN {X 0,Y 284.632,Z 345.333,A -85,B 0,C 180,E1 -17271.651,E2 -17271.651} C_VEL
LIN {X 0,Y 283.951,Z 345.429,A -85,B 0,C 180,E1 -17272.83,E2 -17272.83} C_VEL
LIN {X 0,Y 281.096,Z 345.774,A -85,B 0,C 180,E1 -17274.752,E2 -17274.752} C_VEL
LIN {X 0,Y 278.725,Z 346.069,A -85,B 0,C 180,E1 -17276.313,E2 -17276.313} C_VEL
LIN {X 0,Y 277.769,Z 346.197,A -85,B 0,C 180,E1 -17277.523,E2 -17277.523} C_VEL
LIN {X 0,Y 277.723,Z 346.199,A -85,B 0,C 180,E1 -17277.932,E2 -17277.932} C_VEL
LIN {X 0,Y 277.849,Z 346.174,A -85,B 0,C 180,E1 -17279.999,E2 -17279.999} C_VEL
LIN {X 0,Y 277.695,Z 346.208,A -85,B 0,C 180,E1 -17282.901,E2 -17282.901} C_VEL
LIN {X 0,Y 277.632,Z 346.214,A -85,B 0,C 180,E1 -17287.271,E2 -17287.271} C_VEL
LIN {X 0,Y 277.485,Z 346.235,A -85,B 0,C 180,E1 -17290.212,E2 -17290.212} C_VEL
LIN {X 0,Y 277.413,Z 346.242,A -85,B 0,C 180,E1 -17294.675,E2 -17294.675} C_VEL
LIN {X 0,Y 277.355,Z 346.25,A -85,B 0,C 180,E1 -17299.232,E2 -17299.232} C_VEL
LIN {X 0,Y 277.327,Z 346.305,A -85,B 0,C 180,E1 -17301.363,E2 -17301.363} C_VEL
LIN {X 0,Y 279.116,Z 352.899,A -85,B 0,C 180,E1 -17305.343,E2 -17305.343} C_VEL
LIN {X 0,Y 280.969,Z 359.861,A -85,B 0,C 180,E1 -17309.192,E2 -17309.192} C_VEL
LIN {X 0,Y 283.491,Z 369.18,A -85,B 0,C 180,E1 -17313.903,E2 -17313.903} C_VEL
LIN {X 0,Y 285.351,Z 376.076,A -85,B 0,C 180,E1 -17317.114,E2 -17317.114} C_VEL
LIN {X 0,Y 287.661,Z 384.486,A -85,B 0,C 180,E1 -17320.773,E2 -17320.773} C_VEL
LIN {X 0,Y 290.7,Z 395.119,A -85,B 0,C 180,E1 -17325.064,E2 -17325.064} C_VEL
LIN {X 0,Y 293.226,Z 405.19,A -85,B 0,C 180,E1 -17328.773,E2 -17328.773} C_VEL
LIN {X 0,Y 291.36,Z 411.512,A -85,B 0,C 180,E1 -17330.72,E2 -17330.72} C_VEL
LIN {X 0,Y 294.186,Z 435.721,A -85,B 0,C 180,E1 -17332.069,E2 -17332.069} C_VEL
LIN {X 0,Y 296.135,Z 452.388,A -85,B 0,C 180,E1 -17333.262,E2 -17333.262} C_VEL
LIN {X 0,Y 297.556,Z 468.646,A -85,B 0,C 180,E1 -17334.654,E2 -17334.654} C_VEL
LIN {X 0,Y 297.651,Z 473.35,A -85,B 0,C 180,E1 -17335.077,E2 -17335.077} C_VEL
LIN {X 0,Y 294.909,Z 489.006,A -85,B 0,C 180,E1 -17336.52,E2 -17336.52} C_VEL
LIN {X 0,Y 291.961,Z 503.996,A -85,B 0,C 180,E1 -17338.231,E2 -17338.231} C_VEL
LIN {X 0,Y 289.341,Z 516.363,A -85,B 0,C 180,E1 -17339.94,E2 -17339.94} C_VEL
LIN {X 0,Y 286.623,Z 528.766,A -85,B 0,C 180,E1 -17341.971,E2 -17341.971} C_VEL
LIN {X 0,Y 283.93,Z 540.86,A -85,B 0,C 180,E1 -17344.336,E2 -17344.336} C_VEL
LIN {X 0,Y 281.54,Z 551.773,A -85,B 0,C 180,E1 -17346.892,E2 -17346.892} C_VEL
LIN {X 0,Y 279.696,Z 560.81,A -85,B 0,C 180,E1 -17349.408,E2 -17349.408} C_VEL
LIN {X 0,Y 278.2,Z 569.575,A -85,B 0,C 180,E1 -17352.357,E2 -17352.357} C_VEL
LIN {X 0,Y 277.128,Z 576.719,A -85,B 0,C 180,E1 -17355.313,E2 -17355.313} C_VEL
LIN {X 0,Y 276.568,Z 582.471,A -85,B 0,C 180,E1 -17358.274,E2 -17358.274} C_VEL
LIN {X 0,Y 276.4,Z 586.947,A -85,B 0,C 180,E1 -17361.228,E2 -17361.228} C_VEL
LIN {X 0,Y 276.458,Z 588.727,A -85,B 0,C 180,E1 -17362.701,E2 -17362.701} C_VEL
LIN {X 0,Y 276.565,Z 591.274,A -85,B 0,C 180,E1 -17365.631,E2 -17365.631} C_VEL
LIN {X 0,Y 276.59,Z 592.658,A -85,B 0,C 180,E1 -17368.548,E2 -17368.548} C_VEL
LIN {X 0,Y 276.596,Z 592.937,A -85,B 0,C 180,E1 -17370.004,E2 -17370.004} C_VEL
LIN {X 0,Y 276.531,Z 592.538,A -85,B 0,C 180,E1 -17372.917,E2 -17372.917} C_VEL
LIN {X 0,Y 276.559,Z 591.942,A -85,B 0,C 180,E1 -17374.376,E2 -17374.376} C_VEL
LIN {X 0,Y 276.291,Z 589.903,A -85,B 0,C 180,E1 -17377.31,E2 -17377.31} C_VEL
LIN {X 0,Y 276.236,Z 586.701,A -85,B 0,C 180,E1 -17380.262,E2 -17380.262} C_VEL
LIN {X 0,Y 276.584,Z 582.496,A -85,B 0,C 180,E1 -17383.223,E2 -17383.223} C_VEL
LIN {X 0,Y 277.356,Z 577.14,A -85,B 0,C 180,E1 -17386.188,E2 -17386.188} C_VEL
LIN {X 0,Y 278.693,Z 570.674,A -85,B 0,C 180,E1 -17389.14,E2 -17389.14} C_VEL
LIN {X 0,Y 280.692,Z 562.923,A -85,B 0,C 180,E1 -17392.12,E2 -17392.12} C_VEL
LIN {X 0,Y 283.657,Z 552.967,A -85,B 0,C 180,E1 -17395.305,E2 -17395.305} C_VEL
LIN {X 0,Y 287.707,Z 541.177,A -85,B 0,C 180,E1 -17398.432,E2 -17398.432} C_VEL
LIN {X 0,Y 292.059,Z 528.889,A -85,B 0,C 180,E1 -17401.159,E2 -17401.159} C_VEL
LIN {X 0,Y 297.258,Z 514.819,A -85,B 0,C 180,E1 -17403.755,E2 -17403.755} C_VEL
LIN {X 0,Y 302.864,Z 499.579,A -85,B 0,C 180,E1 -17406.077,E2 -17406.077} C_VEL
LIN {X 0,Y 308.389,Z 484.325,A -85,B 0,C 180,E1 -17407.978,E2 -17407.978} C_VEL
LIN {X 0,Y 310.039,Z 479.253,A -85,B 0,C 180,E1 -17408.566,E2 -17408.566} C_VEL
LIN {X 0,Y 312.884,Z 466.14,A -85,B 0,C 180,E1 -17410.274,E2 -17410.274} C_VEL
LIN {X 0,Y 315.022,Z 455.543,A -85,B 0,C 180,E1 -17411.6,E2 -17411.6} C_VEL
LIN {X 0,Y 316.554,Z 444.011,A -85,B 0,C 180,E1 -17413.281,E2 -17413.281} C_VEL
LIN {X 0,Y 317.138,Z 437.517,A -85,B 0,C 180,E1 -17414.384,E2 -17414.384} C_VEL
LIN {X 0,Y 316.407,Z 435.285,A -85,B 0,C 180,E1 -17415.302,E2 -17415.302} C_VEL
LIN {X 0,Y 314.663,Z 432.206,A -85,B 0,C 180,E1 -17417.484,E2 -17417.484} C_VEL
LIN {X 0,Y 313.716,Z 430.6,A -85,B 0,C 180,E1 -17419.616,E2 -17419.616} C_VEL
LIN {X 0,Y 313.442,Z 430.272,A -85,B 0,C 180,E1 -17421.111,E2 -17421.111} C_VEL
LIN {X 0,Y 313.225,Z 431.22,A -85,B 0,C 180,E1 -17422.713,E2 -17422.713} C_VEL
LIN {X 0,Y 313.227,Z 433.147,A -85,B 0,C 180,E1 -17424.313,E2 -17424.313} C_VEL
LIN {X 0,Y 313.437,Z 437.817,A -85,B 0,C 180,E1 -17426.856,E2 -17426.856} C_VEL
LIN {X 0,Y 313.819,Z 443.162,A -85,B 0,C 180,E1 -17428.997,E2 -17428.997} C_VEL
LIN {X 0,Y 313.997,Z 448.646,A -85,B 0,C 180,E1 -17430.803,E2 -17430.803} C_VEL
LIN {X 0,Y 313.908,Z 449.948,A -85,B 0,C 180,E1 -17431.153,E2 -17431.153} C_VEL
LIN {X 0,Y 308.957,Z 461.653,A -85,B 0,C 180,E1 -17432.939,E2 -17432.939} C_VEL
LIN {X 0,Y 303.966,Z 472.806,A -85,B 0,C 180,E1 -17435.042,E2 -17435.042} C_VEL
LIN {X 0,Y 299.514,Z 482.258,A -85,B 0,C 180,E1 -17437.222,E2 -17437.222} C_VEL
LIN {X 0,Y 294.996,Z 491.209,A -85,B 0,C 180,E1 -17439.791,E2 -17439.791} C_VEL
LIN {X 0,Y 291.089,Z 498.427,A -85,B 0,C 180,E1 -17442.435,E2 -17442.435} C_VEL
LIN {X 0,Y 288.489,Z 502.774,A -85,B 0,C 180,E1 -17444.457,E2 -17444.457} C_VEL
LIN {X 0,Y 285.494,Z 507.251,A -85,B 0,C 180,E1 -17447.2,E2 -17447.2} C_VEL
LIN {X 0,Y 283.137,Z 510.157,A -85,B 0,C 180,E1 -17449.994,E2 -17449.994} C_VEL
LIN {X 0,Y 281.402,Z 511.533,A -85,B 0,C 180,E1 -17452.827,E2 -17452.827} C_VEL
LIN {X 0,Y 280.029,Z 511.466,A -85,B 0,C 180,E1 -17455.683,E2 -17455.683} C_VEL
LIN {X 0,Y 279.398,Z 510.881,A -85,B 0,C 180,E1 -17457.117,E2 -17457.117} C_VEL
LIN {X 0,Y 278.947,Z 509.89,A -85,B 0,C 180,E1 -17458.557,E2 -17458.557} C_VEL
LIN {X 0,Y 278.583,Z 508.482,A -85,B 0,C 180,E1 -17460.001,E2 -17460.001} C_VEL
LIN {X 0,Y 278.329,Z 505.596,A -85,B 0,C 180,E1 -17462.171,E2 -17462.171} C_VEL
LIN {X 0,Y 278.366,Z 501.744,A -85,B 0,C 180,E1 -17464.344,E2 -17464.344} C_VEL
LIN {X 0,Y 278.314,Z 496.913,A -85,B 0,C 180,E1 -17466.525,E2 -17466.525} C_VEL
LIN {X 0,Y 278.977,Z 489.868,A -85,B 0,C 180,E1 -17469.06,E2 -17469.06} C_VEL
LIN {X 0,Y 279.637,Z 481.128,A -85,B 0,C 180,E1 -17471.6,E2 -17471.6} C_VEL
LIN {X 0,Y 280.689,Z 470.453,A -85,B 0,C 180,E1 -17474.131,E2 -17474.131} C_VEL
LIN {X 0,Y 281.82,Z 459.295,A -85,B 0,C 180,E1 -17476.294,E2 -17476.294} C_VEL
LIN {X 0,Y 283.225,Z 447.072,A -85,B 0,C 180,E1 -17478.258,E2 -17478.258} C_VEL
LIN {X 0,Y 284.579,Z 433.752,A -85,B 0,C 180,E1 -17480.034,E2 -17480.034} C_VEL
LIN {X 0,Y 285.999,Z 419.107,A -85,B 0,C 180,E1 -17481.63,E2 -17481.63} C_VEL
LIN {X 0,Y 286.534,Z 414.161,A -85,B 0,C 180,E1 -17482.087,E2 -17482.087} C_VEL
LIN {X 0,Y 285.666,Z 408.562,A -85,B 0,C 180,E1 -17482.661,E2 -17482.661} C_VEL
LIN {X 0,Y 282.633,Z 394.063,A -85,B 0,C 180,E1 -17484.026,E2 -17484.026} C_VEL
LIN {X 0,Y 278.482,Z 377.145,A -85,B 0,C 180,E1 -17485.369,E2 -17485.369} C_VEL
LIN {X 0,Y 278.065,Z 375.307,A -85,B 0,C 180,E1 -17485.547,E2 -17485.547} C_VEL
LIN {X 0,Y 278.571,Z 369.389,A -85,B 0,C 180,E1 -17489.47,E2 -17489.47} C_VEL
LIN {X 0,Y 279.067,Z 363.129,A -85,B 0,C 180,E1 -17493.787,E2 -17493.787} C_VEL
LIN {X 0,Y 279.233,Z 359.524,A -85,B 0,C 180,E1 -17496.346,E2 -17496.346} C_VEL
LIN {X 0,Y 278.981,Z 355.906,A -85,B 0,C 180,E1 -17499.036,E2 -17499.036} C_VEL
LIN {X 0,Y 278.5,Z 352.895,A -85,B 0,C 180,E1 -17501.486,E2 -17501.486} C_VEL
LIN {X 0,Y 279.952,Z 356.757,A -85,B 0,C 180,E1 -17503.704,E2 -17503.704} C_VEL
LIN {X 0,Y 281.483,Z 363.92,A -85,B 0,C 180,E1 -17507.61,E2 -17507.61} C_VEL
LIN {X 0,Y 282.588,Z 369.739,A -85,B 0,C 180,E1 -17510.768,E2 -17510.768} C_VEL
LIN {X 0,Y 283.052,Z 374.826,A -85,B 0,C 180,E1 -17513.42,E2 -17513.42} C_VEL
LIN {X 0,Y 282.803,Z 383.674,A -85,B 0,C 180,E1 -17517.667,E2 -17517.667} C_VEL
LIN {X 0,Y 282.696,Z 392.72,A -85,B 0,C 180,E1 -17521.81,E2 -17521.81} C_VEL
LIN {X 0,Y 282.874,Z 398.101,A -85,B 0,C 180,E1 -17524.079,E2 -17524.079} C_VEL
LIN {X 0,Y 287.603,Z 410.968,A -85,B 0,C 180,E1 -17525.07,E2 -17525.07} C_VEL
LIN {X 0,Y 290.87,Z 422.504,A -85,B 0,C 180,E1 -17526.141,E2 -17526.141} C_VEL
LIN {X 0,Y 289.899,Z 435.07,A -85,B 0,C 180,E1 -17527.174,E2 -17527.174} C_VEL
LIN {X 0,Y 288.617,Z 446.64,A -85,B 0,C 180,E1 -17528.429,E2 -17528.429} C_VEL
LIN {X 0,Y 287.166,Z 457.582,A -85,B 0,C 180,E1 -17529.96,E2 -17529.96} C_VEL
LIN {X 0,Y 285.885,Z 465.732,A -85,B 0,C 180,E1 -17531.359,E2 -17531.359} C_VEL
LIN {X 0,Y 284.372,Z 474.193,A -85,B 0,C 180,E1 -17533.115,E2 -17533.115} C_VEL
LIN {X 0,Y 282.771,Z 482.411,A -85,B 0,C 180,E1 -17535.238,E2 -17535.238} C_VEL
LIN {X 0,Y 281.813,Z 487.961,A -85,B 0,C 180,E1 -17537.026,E2 -17537.026} C_VEL
LIN {X 0,Y 280.551,Z 493.393,A -85,B 0,C 180,E1 -17539.168,E2 -17539.168} C_VEL
LIN {X 0,Y 279.371,Z 497.675,A -85,B 0,C 180,E1 -17541.315,E2 -17541.315} C_VEL
LIN {X 0,Y 278.946,Z 499.895,A -85,B 0,C 180,E1 -17542.76,E2 -17542.76} C_VEL
LIN {X 0,Y 278.757,Z 501.68,A -85,B 0,C 180,E1 -17544.209,E2 -17544.209} C_VEL
LIN {X 0,Y 278.425,Z 503.07,A -85,B 0,C 180,E1 -17545.654,E2 -17545.654} C_VEL
LIN {X 0,Y 278.056,Z 504.642,A -85,B 0,C 180,E1 -17548.548,E2 -17548.548} C_VEL
LIN {X 0,Y 278.025,Z 504.869,A -85,B 0,C 180,E1 -17549.996,E2 -17549.996} C_VEL
LIN {X 0,Y 278.137,Z 504.114,A -85,B 0,C 180,E1 -17552.893,E2 -17552.893} C_VEL
LIN {X 0,Y 278.434,Z 503.156,A -85,B 0,C 180,E1 -17554.339,E2 -17554.339} C_VEL
LIN {X 0,Y 278.761,Z 501.817,A -85,B 0,C 180,E1 -17555.784,E2 -17555.784} C_VEL
LIN {X 0,Y 279.179,Z 499.04,A -85,B 0,C 180,E1 -17557.955,E2 -17557.955} C_VEL
LIN {X 0,Y 280.108,Z 495.205,A -85,B 0,C 180,E1 -17560.112,E2 -17560.112} C_VEL
LIN {X 0,Y 281.352,Z 490.217,A -85,B 0,C 180,E1 -17562.255,E2 -17562.255} C_VEL
LIN {X 0,Y 282.509,Z 483.975,A -85,B 0,C 180,E1 -17564.401,E2 -17564.401} C_VEL
LIN {X 0,Y 284.046,Z 476.175,A -85,B 0,C 180,E1 -17566.527,E2 -17566.527} C_VEL
LIN {X 0,Y 285.508,Z 468.183,A -85,B 0,C 180,E1 -17568.287,E2 -17568.287} C_VEL
LIN {X 0,Y 286.896,Z 459.452,A -85,B 0,C 180,E1 -17569.866,E2 -17569.866} C_VEL
LIN {X 0,Y 288.348,Z 448.607,A -85,B 0,C 180,E1 -17571.44,E2 -17571.44} C_VEL
LIN {X 0,Y 289.658,Z 438.144,A -85,B 0,C 180,E1 -17572.633,E2 -17572.633} C_VEL
LIN {X 0,Y 290.643,Z 427.124,A -85,B 0,C 180,E1 -17573.626,E2 -17573.626} C_VEL
LIN {X 0,Y 290.89,Z 422.245,A -85,B 0,C 180,E1 -17573.995,E2 -17573.995} C_VEL
LIN {X 0,Y 287.519,Z 410.73,A -85,B 0,C 180,E1 -17575.07,E2 -17575.07} C_VEL
LIN {X 0,Y 282.83,Z 397.94,A -85,B 0,C 180,E1 -17576.064,E2 -17576.064} C_VEL
LIN {X 0,Y 282.761,Z 387.623,A -85,B 0,C 180,E1 -17580.627,E2 -17580.627} C_VEL
LIN {X 0,Y 282.987,Z 378.477,A -85,B 0,C 180,E1 -17584.959,E2 -17584.959} C_VEL
LIN {X 0,Y 283.048,Z 373.57,A -85,B 0,C 180,E1 -17587.386,E2 -17587.386} C_VEL
LIN {X 0,Y 282.284,Z 368.065,A -85,B 0,C 180,E1 -17590.334,E2 -17590.334} C_VEL
LIN {X 0,Y 281.157,Z 362.164,A -85,B 0,C 180,E1 -17593.538,E2 -17593.538} C_VEL
LIN {X 0,Y 279.837,Z 356.126,A -85,B 0,C 180,E1 -17596.739,E2 -17596.739} C_VEL
LIN {X 0,Y 278.007,Z 348.852,A -85,B 0,C 180,E1 -17600.802,E2 -17600.802} C_VEL
LIN {X 0,Y 277.308,Z 346.252,A -85,B 0,C 180,E1 -17602.379,E2 -17602.379} C_VEL
LIN {X 0,Y 277.238,Z 346.263,A -85,B 0,C 180,E1 -17606.102,E2 -17606.102} C_VEL
LIN {X 0,Y 277.244,Z 346.257,A -85,B 0,C 180,E1 -17609.536,E2 -17609.536} C_VEL
LIN {X 0,Y 277.34,Z 346.243,A -85,B 0,C 180,E1 -17612.862,E2 -17612.862} C_VEL
LIN {X 0,Y 277.358,Z 346.244,A -85,B 0,C 180,E1 -17616.082,E2 -17616.082} C_VEL
LIN {X 0,Y 277.356,Z 346.239,A -85,B 0,C 180,E1 -17620.766,E2 -17620.766} C_VEL
LIN {X 0,Y 277.408,Z 346.228,A -85,B 0,C 180,E1 -17625.324,E2 -17625.324} C_VEL
LIN {X 0,Y 277.486,Z 346.22,A -85,B 0,C 180,E1 -17629.787,E2 -17629.787} C_VEL
LIN {X 0,Y 277.63,Z 346.215,A -85,B 0,C 180,E1 -17632.728,E2 -17632.728} C_VEL
LIN {X 0,Y 277.723,Z 346.199,A -85,B 0,C 180,E1 -17637.932,E2 -17637.932} C_VEL
LIN {X 0,Y 277.131,Z 346.276,A -85,B 0,C 180,E1 -17639.143,E2 -17639.143} C_VEL
LIN {X 0,Y 275.556,Z 346.473,A -85,B 0,C 180,E1 -17640.331,E2 -17640.331} C_VEL
LIN {X 0,Y 271.705,Z 346.951,A -85,B 0,C 180,E1 -17642.714,E2 -17642.714} C_VEL
LIN {X 0,Y 270.551,Z 347.097,A -85,B 0,C 180,E1 -17643.958,E2 -17643.958} C_VEL
LIN {X 0,Y 270.426,Z 347.11,A -85,B 0,C 180,E1 -17644.38,E2 -17644.38} C_VEL
LIN {X 0,Y 270.59,Z 347.092,A -85,B 0,C 180,E1 -17647.461,E2 -17647.461} C_VEL
LIN {X 0,Y 270.42,Z 347.115,A -85,B 0,C 180,E1 -17650.481,E2 -17650.481} C_VEL
LIN {X 0,Y 270.381,Z 347.117,A -85,B 0,C 180,E1 -17655.065,E2 -17655.065} C_VEL
LIN {X 0,Y 270.345,Z 347.244,A -85,B 0,C 180,E1 -17660.18,E2 -17660.18} C_VEL
LIN {X 0,Y 272.09,Z 354.03,A -85,B 0,C 180,E1 -17664.41,E2 -17664.41} C_VEL
LIN {X 0,Y 273.919,Z 360.892,A -85,B 0,C 180,E1 -17668.336,E2 -17668.336} C_VEL
LIN {X 0,Y 275.952,Z 368.484,A -85,B 0,C 180,E1 -17672.332,E2 -17672.332} C_VEL
LIN {X 0,Y 278.064,Z 376.058,A -85,B 0,C 180,E1 -17676.03,E2 -17676.03} C_VEL
LIN {X 0,Y 280.309,Z 384.265,A -85,B 0,C 180,E1 -17679.742,E2 -17679.742} C_VEL
LIN {X 0,Y 283.425,Z 395.603,A -85,B 0,C 180,E1 -17684.467,E2 -17684.467} C_VEL
LIN {X 0,Y 285.918,Z 404.872,A -85,B 0,C 180,E1 -17688.018,E2 -17688.018} C_VEL
LIN {X 0,Y 286.177,Z 406.122,A -85,B 0,C 180,E1 -17688.471,E2 -17688.471} C_VEL
LIN {X 0,Y 285.671,Z 408.51,A -85,B 0,C 180,E1 -17689.247,E2 -17689.247} C_VEL
LIN {X 0,Y 284.759,Z 411.312,A -85,B 0,C 180,E1 -17690.122,E2 -17690.122} C_VEL
LIN {X 0,Y 287.227,Z 433.239,A -85,B 0,C 180,E1 -17691.332,E2 -17691.332} C_VEL
LIN {X 0,Y 289.037,Z 449.015,A -85,B 0,C 180,E1 -17692.449,E2 -17692.449} C_VEL
LIN {X 0,Y 290.486,Z 464.226,A -85,B 0,C 180,E1 -17693.739,E2 -17693.739} C_VEL
LIN {X 0,Y 291.015,Z 473.036,A -85,B 0,C 180,E1 -17694.583,E2 -17694.583} C_VEL
LIN {X 0,Y 288.51,Z 487.324,A -85,B 0,C 180,E1 -17695.93,E2 -17695.93} C_VEL
LIN {X 0,Y 285.502,Z 502.138,A -85,B 0,C 180,E1 -17697.634,E2 -17697.634} C_VEL
LIN {X 0,Y 282.828,Z 514.677,A -85,B 0,C 180,E1 -17699.381,E2 -17699.381} C_VEL
LIN {X 0,Y 279.893,Z 527.515,A -85,B 0,C 180,E1 -17701.51,E2 -17701.51} C_VEL
LIN {X 0,Y 276.999,Z 540.2,A -85,B 0,C 180,E1 -17704.049,E2 -17704.049} C_VEL
LIN {X 0,Y 274.583,Z 550.922,A -85,B 0,C 180,E1 -17706.631,E2 -17706.631} C_VEL
LIN {X 0,Y 272.694,Z 560.064,A -85,B 0,C 180,E1 -17709.249,E2 -17709.249} C_VEL
LIN {X 0,Y 271.344,Z 567.763,A -85,B 0,C 180,E1 -17711.896,E2 -17711.896} C_VEL
LIN {X 0,Y 270.186,Z 575.061,A -85,B 0,C 180,E1 -17714.927,E2 -17714.927} C_VEL
LIN {X 0,Y 269.572,Z 580.949,A -85,B 0,C 180,E1 -17717.966,E2 -17717.966} C_VEL
LIN {X 0,Y 269.404,Z 585.542,A -85,B 0,C 180,E1 -17720.999,E2 -17720.999} C_VEL
LIN {X 0,Y 269.469,Z 588.797,A -85,B 0,C 180,E1 -17724.016,E2 -17724.016} C_VEL
LIN {X 0,Y 269.587,Z 590.866,A -85,B 0,C 180,E1 -17727.015,E2 -17727.015} C_VEL
LIN {X 0,Y 269.596,Z 591.745,A -85,B 0,C 180,E1 -17730.004,E2 -17730.004} C_VEL
LIN {X 0,Y 269.512,Z 591.413,A -85,B 0,C 180,E1 -17732.993,E2 -17732.993} C_VEL
LIN {X 0,Y 269.527,Z 590.857,A -85,B 0,C 180,E1 -17734.49,E2 -17734.49} C_VEL
LIN {X 0,Y 269.231,Z 588.842,A -85,B 0,C 180,E1 -17737.503,E2 -17737.503} C_VEL
LIN {X 0,Y 269.171,Z 585.725,A -85,B 0,C 180,E1 -17740.534,E2 -17740.534} C_VEL
LIN {X 0,Y 269.576,Z 581.609,A -85,B 0,C 180,E1 -17743.574,E2 -17743.574} C_VEL
LIN {X 0,Y 270.423,Z 576.328,A -85,B 0,C 180,E1 -17746.615,E2 -17746.615} C_VEL
LIN {X 0,Y 271.849,Z 570.017,A -85,B 0,C 180,E1 -17749.642,E2 -17749.642} C_VEL
LIN {X 0,Y 274.245,Z 561.531,A -85,B 0,C 180,E1 -17753.008,E2 -17753.008} C_VEL
LIN {X 0,Y 277.572,Z 551.478,A -85,B 0,C 180,E1 -17756.305,E2 -17756.305} C_VEL
LIN {X 0,Y 282.06,Z 539.488,A -85,B 0,C 180,E1 -17759.55,E2 -17759.55} C_VEL
LIN {X 0,Y 286.592,Z 527.648,A -85,B 0,C 180,E1 -17762.237,E2 -17762.237} C_VEL
LIN {X 0,Y 292.152,Z 513.843,A -85,B 0,C 180,E1 -17764.846,E2 -17764.846} C_VEL
LIN {X 0,Y 298.137,Z 498.956,A -85,B 0,C 180,E1 -17767.164,E2 -17767.164} C_VEL
LIN {X 0,Y 304.832,Z 481.664,A -85,B 0,C 180,E1 -17769.351,E2 -17769.351} C_VEL
LIN {X 0,Y 308.201,Z 468.72,A -85,B 0,C 180,E1 -17771.137,E2 -17771.137} C_VEL
LIN {X 0,Y 310.811,Z 457.936,A -85,B 0,C 180,E1 -17772.558,E2 -17772.558} C_VEL
LIN {X 0,Y 312.855,Z 446.424,A -85,B 0,C 180,E1 -17774.341,E2 -17774.341} C_VEL
LIN {X 0,Y 313.336,Z 443.46,A -85,B 0,C 180,E1 -17774.859,E2 -17774.859} C_VEL
LIN {X 0,Y 313.2,Z 441.768,A -85,B 0,C 180,E1 -17775.382,E2 -17775.382} C_VEL
LIN {X 0,Y 311.649,Z 438.77,A -85,B 0,C 180,E1 -17777.428,E2 -17777.428} C_VEL
LIN {X 0,Y 310.847,Z 437.372,A -85,B 0,C 180,E1 -17779.03,E2 -17779.03} C_VEL
LIN {X 0,Y 310.401,Z 436.756,A -85,B 0,C 180,E1 -17780.657,E2 -17780.657} C_VEL
LIN {X 0,Y 309.998,Z 437.454,A -85,B 0,C 180,E1 -17782.516,E2 -17782.516} C_VEL
LIN {X 0,Y 309.809,Z 438.883,A -85,B 0,C 180,E1 -17783.857,E2 -17783.857} C_VEL
LIN {X 0,Y 309.601,Z 442.989,A -85,B 0,C 180,E1 -17786.246,E2 -17786.246} C_VEL
LIN {X 0,Y 309.612,Z 446.527,A -85,B 0,C 180,E1 -17787.879,E2 -17787.879} C_VEL
LIN {X 0,Y 309.436,Z 452.418,A -85,B 0,C 180,E1 -17790.022,E2 -17790.022} C_VEL
LIN {X 0,Y 309.338,Z 453.339,A -85,B 0,C 180,E1 -17790.319,E2 -17790.319} C_VEL
LIN {X 0,Y 304.207,Z 464.489,A -85,B 0,C 180,E1 -17792.107,E2 -17792.107} C_VEL
LIN {X 0,Y 298.94,Z 475.277,A -85,B 0,C 180,E1 -17794.22,E2 -17794.22} C_VEL
LIN {X 0,Y 294.204,Z 484.456,A -85,B 0,C 180,E1 -17796.414,E2 -17796.414} C_VEL
LIN {X 0,Y 289.983,Z 492.162,A -85,B 0,C 180,E1 -17798.683,E2 -17798.683} C_VEL
LIN {X 0,Y 285.697,Z 499.392,A -85,B 0,C 180,E1 -17801.35,E2 -17801.35} C_VEL
LIN {X 0,Y 281.998,Z 505.076,A -85,B 0,C 180,E1 -17804.09,E2 -17804.09} C_VEL
LIN {X 0,Y 278.846,Z 509.229,A -85,B 0,C 180,E1 -17806.89,E2 -17806.89} C_VEL
LIN {X 0,Y 276.37,Z 511.878,A -85,B 0,C 180,E1 -17809.747,E2 -17809.747} C_VEL
LIN {X 0,Y 274.533,Z 513.051,A -85,B 0,C 180,E1 -17812.647,E2 -17812.647} C_VEL
LIN {X 0,Y 273.085,Z 512.781,A -85,B 0,C 180,E1 -17815.573,E2 -17815.573} C_VEL
LIN {X 0,Y 272.413,Z 512.099,A -85,B 0,C 180,E1 -17817.043,E2 -17817.043} C_VEL
LIN {X 0,Y 271.564,Z 509.468,A -85,B 0,C 180,E1 -17820.001,E2 -17820.001} C_VEL
LIN {X 0,Y 271.297,Z 506.463,A -85,B 0,C 180,E1 -17822.228,E2 -17822.228} C_VEL
LIN {X 0,Y 271.324,Z 502.469,A -85,B 0,C 180,E1 -17824.457,E2 -17824.457} C_VEL
LIN {X 0,Y 271.276,Z 497.487,A -85,B 0,C 180,E1 -17826.695,E2 -17826.695} C_VEL
LIN {X 0,Y 271.996,Z 490.276,A -85,B 0,C 180,E1 -17829.294,E2 -17829.294} C_VEL
LIN {X 0,Y 272.657,Z 481.321,A -85,B 0,C 180,E1 -17831.901,E2 -17831.901} C_VEL
LIN {X 0,Y 273.609,Z 472.087,A -85,B 0,C 180,E1 -17834.125,E2 -17834.125} C_VEL
LIN {X 0,Y 274.747,Z 461.086,A -85,B 0,C 180,E1 -17836.343,E2 -17836.343} C_VEL
LIN {X 0,Y 276.305,Z 447.866,A -85,B 0,C 180,E1 -17838.539,E2 -17838.539} C_VEL
LIN {X 0,Y 277.743,Z 434.225,A -85,B 0,C 180,E1 -17840.395,E2 -17840.395} C_VEL
LIN {X 0,Y 279.154,Z 419.868,A -85,B 0,C 180,E1 -17841.994,E2 -17841.994} C_VEL
LIN {X 0,Y 279.62,Z 413.716,A -85,B 0,C 180,E1 -17842.589,E2 -17842.589} C_VEL
LIN {X 0,Y 276.365,Z 397.817,A -85,B 0,C 180,E1 -17844.195,E2 -17844.195} C_VEL
LIN {X 0,Y 272.779,Z 382.383,A -85,B 0,C 180,E1 -17845.517,E2 -17845.517} C_VEL
LIN {X 0,Y 271.125,Z 375.737,A -85,B 0,C 180,E1 -17846.05,E2 -17846.05} C_VEL
LIN {X 0,Y 271.663,Z 369.478,A -85,B 0,C 180,E1 -17850.297,E2 -17850.297} C_VEL
LIN {X 0,Y 272.211,Z 363.306,A -85,B 0,C 180,E1 -17854.612,E2 -17854.612} C_VEL
LIN {X 0,Y 272.267,Z 360.245,A -85,B 0,C 180,E1 -17856.847,E2 -17856.847} C_VEL
LIN {X 0,Y 272.022,Z 357.187,A -85,B 0,C 180,E1 -17859.183,E2 -17859.183} C_VEL
LIN {X 0,Y 271.648,Z 355.117,A -85,B 0,C 180,E1 -17860.904,E2 -17860.904} C_VEL
LIN {X 0,Y 273.085,Z 358.39,A -85,B 0,C 180,E1 -17863,E2 -17863} C_VEL
LIN {X 0,Y 274.434,Z 364.246,A -85,B 0,C 180,E1 -17866.252,E2 -17866.252} C_VEL
LIN {X 0,Y 275.675,Z 370.732,A -85,B 0,C 180,E1 -17869.891,E2 -17869.891} C_VEL
LIN {X 0,Y 276.372,Z 375.465,A -85,B 0,C 180,E1 -17872.385,E2 -17872.385} C_VEL
LIN {X 0,Y 276.218,Z 382.708,A -85,B 0,C 180,E1 -17875.957,E2 -17875.957} C_VEL
LIN {X 0,Y 275.993,Z 391.916,A -85,B 0,C 180,E1 -17880.276,E2 -17880.276} C_VEL
LIN {X 0,Y 276.117,Z 398.981,A -85,B 0,C 180,E1 -17883.391,E2 -17883.391} C_VEL
LIN {X 0,Y 280.957,Z 411.982,A -85,B 0,C 180,E1 -17884.435,E2 -17884.435} C_VEL
LIN {X 0,Y 284.371,Z 423.769,A -85,B 0,C 180,E1 -17885.577,E2 -17885.577} C_VEL
LIN {X 0,Y 283.434,Z 436.13,A -85,B 0,C 180,E1 -17886.623,E2 -17886.623} C_VEL
LIN {X 0,Y 282.101,Z 447.704,A -85,B 0,C 180,E1 -17887.904,E2 -17887.904} C_VEL
LIN {X 0,Y 280.581,Z 458.652,A -85,B 0,C 180,E1 -17889.468,E2 -17889.468} C_VEL
LIN {X 0,Y 279.266,Z 466.801,A -85,B 0,C 180,E1 -17890.9,E2 -17890.9} C_VEL
LIN {X 0,Y 277.678,Z 475.264,A -85,B 0,C 180,E1 -17892.696,E2 -17892.696} C_VEL
LIN {X 0,Y 275.991,Z 483.486,A -85,B 0,C 180,E1 -17894.867,E2 -17894.867} C_VEL
LIN {X 0,Y 274.981,Z 489.037,A -85,B 0,C 180,E1 -17896.698,E2 -17896.698} C_VEL
LIN {X 0,Y 273.662,Z 494.47,A -85,B 0,C 180,E1 -17898.891,E2 -17898.891} C_VEL
LIN {X 0,Y 272.437,Z 498.752,A -85,B 0,C 180,E1 -17901.092,E2 -17901.092} C_VEL
LIN {X 0,Y 271.986,Z 500.972,A -85,B 0,C 180,E1 -17902.573,E2 -17902.573} C_VEL
LIN {X 0,Y 271.775,Z 502.757,A -85,B 0,C 180,E1 -17904.059,E2 -17904.059} C_VEL
LIN {X 0,Y 271.428,Z 504.147,A -85,B 0,C 180,E1 -17905.541,E2 -17905.541} C_VEL
LIN {X 0,Y 271.065,Z 505.716,A -85,B 0,C 180,E1 -17908.511,E2 -17908.511} C_VEL
LIN {X 0,Y 271.027,Z 505.943,A -85,B 0,C 180,E1 -17909.996,E2 -17909.996} C_VEL
LIN {X 0,Y 271.148,Z 505.187,A -85,B 0,C 180,E1 -17912.968,E2 -17912.968} C_VEL
LIN {X 0,Y 271.777,Z 502.893,A -85,B 0,C 180,E1 -17915.933,E2 -17915.933} C_VEL
LIN {X 0,Y 272.228,Z 500.115,A -85,B 0,C 180,E1 -17918.159,E2 -17918.159} C_VEL
LIN {X 0,Y 273.202,Z 496.279,A -85,B 0,C 180,E1 -17920.37,E2 -17920.37} C_VEL
LIN {X 0,Y 274.502,Z 491.29,A -85,B 0,C 180,E1 -17922.566,E2 -17922.566} C_VEL
LIN {X 0,Y 275.716,Z 485.047,A -85,B 0,C 180,E1 -17924.764,E2 -17924.764} C_VEL
LIN {X 0,Y 277.326,Z 477.244,A -85,B 0,C 180,E1 -17926.94,E2 -17926.94} C_VEL
LIN {X 0,Y 278.851,Z 469.25,A -85,B 0,C 180,E1 -17928.74,E2 -17928.74} C_VEL
LIN {X 0,Y 280.308,Z 460.514,A -85,B 0,C 180,E1 -17930.353,E2 -17930.353} C_VEL
LIN {X 0,Y 281.826,Z 449.664,A -85,B 0,C 180,E1 -17931.962,E2 -17931.962} C_VEL
LIN {X 0,Y 283.189,Z 439.175,A -85,B 0,C 180,E1 -17933.182,E2 -17933.182} C_VEL
LIN {X 0,Y 284.346,Z 426.868,A -85,B 0,C 180,E1 -17934.296,E2 -17934.296} C_VEL
LIN {X 0,Y 284.362,Z 423.637,A -85,B 0,C 180,E1 -17934.554,E2 -17934.554} C_VEL
LIN {X 0,Y 280.915,Z 411.874,A -85,B 0,C 180,E1 -17935.696,E2 -17935.696} C_VEL
LIN {X 0,Y 276.107,Z 398.893,A -85,B 0,C 180,E1 -17936.775,E2 -17936.775} C_VEL
LIN {X 0,Y 276.128,Z 388.52,A -85,B 0,C 180,E1 -17941.446,E2 -17941.446} C_VEL
LIN {X 0,Y 276.392,Z 379.4,A -85,B 0,C 180,E1 -17945.786,E2 -17945.786} C_VEL
LIN {X 0,Y 276.316,Z 375.155,A -85,B 0,C 180,E1 -17947.956,E2 -17947.956} C_VEL
LIN {X 0,Y 275.592,Z 370.127,A -85,B 0,C 180,E1 -17950.687,E2 -17950.687} C_VEL
LIN {X 0,Y 274.523,Z 364.587,A -85,B 0,C 180,E1 -17953.721,E2 -17953.721} C_VEL
LIN {X 0,Y 273.246,Z 358.59,A -85,B 0,C 180,E1 -17957.031,E2 -17957.031} C_VEL
LIN {X 0,Y 271.599,Z 351.835,A -85,B 0,C 180,E1 -17960.915,E2 -17960.915} C_VEL
LIN {X 0,Y 270.25,Z 347.131,A -85,B 0,C 180,E1 -17963.716,E2 -17963.716} C_VEL
LIN {X 0,Y 270.187,Z 347.136,A -85,B 0,C 180,E1 -17966.89,E2 -17966.89} C_VEL
LIN {X 0,Y 270.211,Z 347.131,A -85,B 0,C 180,E1 -17970.384,E2 -17970.384} C_VEL
LIN {X 0,Y 270.251,Z 347.124,A -85,B 0,C 180,E1 -17973.762,E2 -17973.762} C_VEL
LIN {X 0,Y 270.252,Z 347.122,A -85,B 0,C 180,E1 -17977.04,E2 -17977.04} C_VEL
LIN {X 0,Y 270.311,Z 347.12,A -85,B 0,C 180,E1 -17980.245,E2 -17980.245} C_VEL
LIN {X 0,Y 270.376,Z 347.107,A -85,B 0,C 180,E1 -17984.933,E2 -17984.933} C_VEL
LIN {X 0,Y 270.421,Z 347.102,A -85,B 0,C 180,E1 -17989.518,E2 -17989.518} C_VEL
LIN {X 0,Y 270.589,Z 347.092,A -85,B 0,C 180,E1 -17992.538,E2 -17992.538} C_VEL
LIN {X 0,Y 270.763,Z 347.071,A -85,B 0,C 180,E1 -17998.512,E2 -17998.512} C_VEL
LIN {X 0,Y 270.771,Z 347.055,A -85,B 0,C 180,E1 -18001.487,E2 -18001.487} C_VEL
LIN {X 0,Y 270.426,Z 347.11,A -85,B 0,C 180,E1 -18004.38,E2 -18004.38} C_VEL
LIN {X 0,Y 269.692,Z 347.207,A -85,B 0,C 180,E1 -18005.624,E2 -18005.624} C_VEL
LIN {X 0,Y 266.863,Z 347.563,A -85,B 0,C 180,E1 -18007.653,E2 -18007.653} C_VEL
LIN {X 0,Y 264.487,Z 347.857,A -85,B 0,C 180,E1 -18009.302,E2 -18009.302} C_VEL
LIN {X 0,Y 263.438,Z 347.984,A -85,B 0,C 180,E1 -18010.579,E2 -18010.579} C_VEL
LIN {X 0,Y 263.333,Z 347.995,A -85,B 0,C 180,E1 -18011.012,E2 -18011.012} C_VEL
LIN {X 0,Y 263.329,Z 347.997,A -85,B 0,C 180,E1 -18015.479,E2 -18015.479} C_VEL
LIN {X 0,Y 263.246,Z 348.084,A -85,B 0,C 180,E1 -18018.887,E2 -18018.887} C_VEL
LIN {X 0,Y 264.755,Z 353.816,A -85,B 0,C 180,E1 -18022.637,E2 -18022.637} C_VEL
LIN {X 0,Y 266.482,Z 360.469,A -85,B 0,C 180,E1 -18026.637,E2 -18026.637} C_VEL
LIN {X 0,Y 268.438,Z 367.801,A -85,B 0,C 180,E1 -18030.698,E2 -18030.698} C_VEL
LIN {X 0,Y 270.678,Z 375.897,A -85,B 0,C 180,E1 -18034.835,E2 -18034.835} C_VEL
LIN {X 0,Y 273.449,Z 386.012,A -85,B 0,C 180,E1 -18039.56,E2 -18039.56} C_VEL
LIN {X 0,Y 276.337,Z 396.595,A -85,B 0,C 180,E1 -18044.076,E2 -18044.076} C_VEL
LIN {X 0,Y 278.765,Z 405.547,A -85,B 0,C 180,E1 -18047.611,E2 -18047.611} C_VEL
LIN {X 0,Y 279.127,Z 407.018,A -85,B 0,C 180,E1 -18048.167,E2 -18048.167} C_VEL
LIN {X 0,Y 278.687,Z 409.576,A -85,B 0,C 180,E1 -18049.035,E2 -18049.035} C_VEL
LIN {X 0,Y 278.247,Z 410.89,A -85,B 0,C 180,E1 -18049.456,E2 -18049.456} C_VEL
LIN {X 0,Y 280.676,Z 434.06,A -85,B 0,C 180,E1 -18050.794,E2 -18050.794} C_VEL
LIN {X 0,Y 282.478,Z 450.694,A -85,B 0,C 180,E1 -18052.033,E2 -18052.033} C_VEL
LIN {X 0,Y 283.836,Z 466.327,A -85,B 0,C 180,E1 -18053.436,E2 -18053.436} C_VEL
LIN {X 0,Y 284.099,Z 474.47,A -85,B 0,C 180,E1 -18054.242,E2 -18054.242} C_VEL
LIN {X 0,Y 281.338,Z 489.118,A -85,B 0,C 180,E1 -18055.692,E2 -18055.692} C_VEL
LIN {X 0,Y 278.494,Z 502.922,A -85,B 0,C 180,E1 -18057.361,E2 -18057.361} C_VEL
LIN {X 0,Y 275.76,Z 515.177,A -85,B 0,C 180,E1 -18059.147,E2 -18059.147} C_VEL
LIN {X 0,Y 272.746,Z 528.192,A -85,B 0,C 180,E1 -18061.408,E2 -18061.408} C_VEL
LIN {X 0,Y 270.07,Z 539.458,A -85,B 0,C 180,E1 -18063.748,E2 -18063.748} C_VEL
LIN {X 0,Y 267.623,Z 550.149,A -85,B 0,C 180,E1 -18066.397,E2 -18066.397} C_VEL
LIN {X 0,Y 265.682,Z 559.253,A -85,B 0,C 180,E1 -18069.082,E2 -18069.082} C_VEL
LIN {X 0,Y 264.122,Z 567.947,A -85,B 0,C 180,E1 -18072.186,E2 -18072.186} C_VEL
LIN {X 0,Y 263.079,Z 575.009,A -85,B 0,C 180,E1 -18075.302,E2 -18075.302} C_VEL
LIN {X 0,Y 262.504,Z 580.65,A -85,B 0,C 180,E1 -18078.421,E2 -18078.421} C_VEL
LIN {X 0,Y 262.42,Z 584.056,A -85,B 0,C 180,E1 -18080.757,E2 -18080.757} C_VEL
LIN {X 0,Y 262.466,Z 587.428,A -85,B 0,C 180,E1 -18083.855,E2 -18083.855} C_VEL
LIN {X 0,Y 262.581,Z 589.602,A -85,B 0,C 180,E1 -18086.935,E2 -18086.935} C_VEL
LIN {X 0,Y 262.628,Z 590.529,A -85,B 0,C 180,E1 -18090.004,E2 -18090.004} C_VEL
LIN {X 0,Y 262.494,Z 590.279,A -85,B 0,C 180,E1 -18093.073,E2 -18093.073} C_VEL
LIN {X 0,Y 262.491,Z 589.764,A -85,B 0,C 180,E1 -18094.611,E2 -18094.611} C_VEL
LIN {X 0,Y 262.17,Z 587.78,A -85,B 0,C 180,E1 -18097.706,E2 -18097.706} C_VEL
LIN {X 0,Y 262.125,Z 584.762,A -85,B 0,C 180,E1 -18100.821,E2 -18100.821} C_VEL
LIN {X 0,Y 262.566,Z 580.692,A -85,B 0,C 180,E1 -18103.943,E2 -18103.943} C_VEL
LIN {X 0,Y 263.484,Z 575.555,A -85,B 0,C 180,E1 -18107.066,E2 -18107.066} C_VEL
LIN {X 0,Y 265.028,Z 569.385,A -85,B 0,C 180,E1 -18110.169,E2 -18110.169} C_VEL
LIN {X 0,Y 267.957,Z 560.064,A -85,B 0,C 180,E1 -18113.991,E2 -18113.991} C_VEL
LIN {X 0,Y 271.622,Z 550.085,A -85,B 0,C 180,E1 -18117.343,E2 -18117.343} C_VEL
LIN {X 0,Y 275.781,Z 539.735,A -85,B 0,C 180,E1 -18120.246,E2 -18120.246} C_VEL
LIN {X 0,Y 280.616,Z 528.13,A -85,B 0,C 180,E1 -18123.009,E2 -18123.009} C_VEL
LIN {X 0,Y 286.412,Z 514.812,A -85,B 0,C 180,E1 -18125.65,E2 -18125.65} C_VEL
LIN {X 0,Y 293.073,Z 499.572,A -85,B 0,C 180,E1 -18128.137,E2 -18128.137} C_VEL
LIN {X 0,Y 300.048,Z 483.116,A -85,B 0,C 180,E1 -18130.323,E2 -18130.323} C_VEL
LIN {X 0,Y 303.829,Z 470.503,A -85,B 0,C 180,E1 -18132.133,E2 -18132.133} C_VEL
LIN {X 0,Y 306.59,Z 461.011,A -85,B 0,C 180,E1 -18133.451,E2 -18133.451} C_VEL
LIN {X 0,Y 308.729,Z 451.994,A -85,B 0,C 180,E1 -18134.889,E2 -18134.889} C_VEL
LIN {X 0,Y 309.554,Z 448.223,A -85,B 0,C 180,E1 -18135.56,E2 -18135.56} C_VEL
LIN {X 0,Y 309.347,Z 447.014,A -85,B 0,C 180,E1 -18136.054,E2 -18136.054} C_VEL
LIN {X 0,Y 307.818,Z 444.066,A -85,B 0,C 180,E1 -18138.539,E2 -18138.539} C_VEL
LIN {X 0,Y 307.213,Z 443.197,A -85,B 0,C 180,E1 -18140.168,E2 -18140.168} C_VEL
LIN {X 0,Y 306.754,Z 443.364,A -85,B 0,C 180,E1 -18141.787,E2 -18141.787} C_VEL
LIN {X 0,Y 306.288,Z 444.699,A -85,B 0,C 180,E1 -18143.431,E2 -18143.431} C_VEL
LIN {X 0,Y 305.674,Z 448.544,A -85,B 0,C 180,E1 -18145.867,E2 -18145.867} C_VEL
LIN {X 0,Y 305.437,Z 451.338,A -85,B 0,C 180,E1 -18147.261,E2 -18147.261} C_VEL
LIN {X 0,Y 304.843,Z 457.172,A -85,B 0,C 180,E1 -18149.523,E2 -18149.523} C_VEL
LIN {X 0,Y 298.762,Z 469.161,A -85,B 0,C 180,E1 -18151.553,E2 -18151.553} C_VEL
LIN {X 0,Y 292.58,Z 480.542,A -85,B 0,C 180,E1 -18154,E2 -18154} C_VEL
LIN {X 0,Y 287.034,Z 490.113,A -85,B 0,C 180,E1 -18156.555,E2 -18156.555} C_VEL
LIN {X 0,Y 281.572,Z 498.794,A -85,B 0,C 180,E1 -18159.548,E2 -18159.548} C_VEL
LIN {X 0,Y 277.415,Z 504.885,A -85,B 0,C 180,E1 -18162.302,E2 -18162.302} C_VEL
LIN {X 0,Y 273.804,Z 509.455,A -85,B 0,C 180,E1 -18165.127,E2 -18165.127} C_VEL
LIN {X 0,Y 270.831,Z 512.578,A -85,B 0,C 180,E1 -18168.019,E2 -18168.019} C_VEL
LIN {X 0,Y 268.542,Z 514.275,A -85,B 0,C 180,E1 -18170.966,E2 -18170.966} C_VEL
LIN {X 0,Y 266.855,Z 514.507,A -85,B 0,C 180,E1 -18173.954,E2 -18173.954} C_VEL
LIN {X 0,Y 266.131,Z 514.07,A -85,B 0,C 180,E1 -18175.457,E2 -18175.457} C_VEL
LIN {X 0,Y 265.419,Z 513.258,A -85,B 0,C 180,E1 -18176.965,E2 -18176.965} C_VEL
LIN {X 0,Y 264.544,Z 510.439,A -85,B 0,C 180,E1 -18180.001,E2 -18180.001} C_VEL
LIN {X 0,Y 264.264,Z 507.262,A -85,B 0,C 180,E1 -18182.287,E2 -18182.287} C_VEL
LIN {X 0,Y 264.282,Z 503.147,A -85,B 0,C 180,E1 -18184.576,E2 -18184.576} C_VEL
LIN {X 0,Y 264.238,Z 498.019,A -85,B 0,C 180,E1 -18186.875,E2 -18186.875} C_VEL
LIN {X 0,Y 264.999,Z 490.573,A -85,B 0,C 180,E1 -18189.542,E2 -18189.542} C_VEL
LIN {X 0,Y 265.698,Z 481.477,A -85,B 0,C 180,E1 -18192.217,E2 -18192.217} C_VEL
LIN {X 0,Y 266.688,Z 472.061,A -85,B 0,C 180,E1 -18194.499,E2 -18194.499} C_VEL
LIN {X 0,Y 267.989,Z 459.749,A -85,B 0,C 180,E1 -18196.964,E2 -18196.964} C_VEL
LIN {X 0,Y 269.541,Z 447.284,A -85,B 0,C 180,E1 -18199.022,E2 -18199.022} C_VEL
LIN {X 0,Y 271.142,Z 432.224,A -85,B 0,C 180,E1 -18201.067,E2 -18201.067} C_VEL
LIN {X 0,Y 272.565,Z 418.75,A -85,B 0,C 180,E1 -18202.554,E2 -18202.554} C_VEL
LIN {X 0,Y 272.874,Z 415.703,A -85,B 0,C 180,E1 -18202.85,E2 -18202.85} C_VEL
LIN {X 0,Y 270.075,Z 401.238,A -85,B 0,C 180,E1 -18204.38,E2 -18204.38} C_VEL
LIN {X 0,Y 266.163,Z 384.238,A -85,B 0,C 180,E1 -18205.91,E2 -18205.91} C_VEL
LIN {X 0,Y 264.173,Z 376.197,A -85,B 0,C 180,E1 -18206.565,E2 -18206.565} C_VEL
LIN {X 0,Y 264.657,Z 370.748,A -85,B 0,C 180,E1 -18210.302,E2 -18210.302} C_VEL
LIN {X 0,Y 265.256,Z 364.461,A -85,B 0,C 180,E1 -18214.775,E2 -18214.775} C_VEL
LIN {X 0,Y 265.251,Z 360.746,A -85,B 0,C 180,E1 -18217.547,E2 -18217.547} C_VEL
LIN {X 0,Y 264.837,Z 357.273,A -85,B 0,C 180,E1 -18220.37,E2 -18220.37} C_VEL
LIN {X 0,Y 266.762,Z 361.827,A -85,B 0,C 180,E1 -18223.235,E2 -18223.235} C_VEL
LIN {X 0,Y 268.196,Z 368.519,A -85,B 0,C 180,E1 -18227.049,E2 -18227.049} C_VEL
LIN {X 0,Y 269.258,Z 374.273,A -85,B 0,C 180,E1 -18230.276,E2 -18230.276} C_VEL
LIN {X 0,Y 269.743,Z 378.038,A -85,B 0,C 180,E1 -18232.337,E2 -18232.337} C_VEL
LIN {X 0,Y 269.567,Z 385.309,A -85,B 0,C 180,E1 -18235.905,E2 -18235.905} C_VEL
LIN {X 0,Y 269.336,Z 394.621,A -85,B 0,C 180,E1 -18240.275,E2 -18240.275} C_VEL
LIN {X 0,Y 269.476,Z 400.185,A -85,B 0,C 180,E1 -18242.686,E2 -18242.686} C_VEL
LIN {X 0,Y 274.265,Z 412.824,A -85,B 0,C 180,E1 -18243.751,E2 -18243.751} C_VEL
LIN {X 0,Y 277.544,Z 424.006,A -85,B 0,C 180,E1 -18244.862,E2 -18244.862} C_VEL
LIN {X 0,Y 278.003,Z 426.116,A -85,B 0,C 180,E1 -18245.087,E2 -18245.087} C_VEL
LIN {X 0,Y 276.998,Z 437.191,A -85,B 0,C 180,E1 -18246.046,E2 -18246.046} C_VEL
LIN {X 0,Y 275.607,Z 448.769,A -85,B 0,C 180,E1 -18247.354,E2 -18247.354} C_VEL
LIN {X 0,Y 274.017,Z 459.722,A -85,B 0,C 180,E1 -18248.953,E2 -18248.953} C_VEL
LIN {X 0,Y 272.646,Z 467.873,A -85,B 0,C 180,E1 -18250.418,E2 -18250.418} C_VEL
LIN {X 0,Y 271.006,Z 476.335,A -85,B 0,C 180,E1 -18252.256,E2 -18252.256} C_VEL
LIN {X 0,Y 269.223,Z 484.562,A -85,B 0,C 180,E1 -18254.477,E2 -18254.477} C_VEL
LIN {X 0,Y 268.155,Z 490.113,A -85,B 0,C 180,E1 -18256.353,E2 -18256.353} C_VEL
LIN {X 0,Y 266.78,Z 495.546,A -85,B 0,C 180,E1 -18258.601,E2 -18258.601} C_VEL
LIN {X 0,Y 265.507,Z 499.829,A -85,B 0,C 180,E1 -18260.858,E2 -18260.858} C_VEL
LIN {X 0,Y 265.028,Z 502.049,A -85,B 0,C 180,E1 -18262.377,E2 -18262.377} C_VEL
LIN {X 0,Y 264.794,Z 503.835,A -85,B 0,C 180,E1 -18263.902,E2 -18263.902} C_VEL
LIN {X 0,Y 264.433,Z 505.224,A -85,B 0,C 180,E1 -18265.423,E2 -18265.423} C_VEL
LIN {X 0,Y 264.07,Z 506.79,A -85,B 0,C 180,E1 -18268.471,E2 -18268.471} C_VEL
LIN {X 0,Y 264.026,Z 507.017,A -85,B 0,C 180,E1 -18269.996,E2 -18269.996} C_VEL
LIN {X 0,Y 264.156,Z 506.261,A -85,B 0,C 180,E1 -18273.046,E2 -18273.046} C_VEL
LIN {X 0,Y 264.794,Z 503.969,A -85,B 0,C 180,E1 -18276.09,E2 -18276.09} C_VEL
LIN {X 0,Y 265.281,Z 501.191,A -85,B 0,C 180,E1 -18278.374,E2 -18278.374} C_VEL
LIN {X 0,Y 266.303,Z 497.353,A -85,B 0,C 180,E1 -18280.642,E2 -18280.642} C_VEL
LIN {X 0,Y 267.66,Z 492.362,A -85,B 0,C 180,E1 -18282.892,E2 -18282.892} C_VEL
LIN {X 0,Y 268.953,Z 486.115,A -85,B 0,C 180,E1 -18285.144,E2 -18285.144} C_VEL
LIN {X 0,Y 270.631,Z 478.311,A -85,B 0,C 180,E1 -18287.372,E2 -18287.372} C_VEL
LIN {X 0,Y 272.212,Z 470.317,A -85,B 0,C 180,E1 -18289.215,E2 -18289.215} C_VEL
LIN {X 0,Y 273.74,Z 461.577,A -85,B 0,C 180,E1 -18290.864,E2 -18290.864} C_VEL
LIN {X 0,Y 275.328,Z 450.721,A -85,B 0,C 180,E1 -18292.508,E2 -18292.508} C_VEL
LIN {X 0,Y 276.756,Z 440.155,A -85,B 0,C 180,E1 -18293.762,E2 -18293.762} C_VEL
LIN {X 0,Y 277.929,Z 428.21,A -85,B 0,C 180,E1 -18294.869,E2 -18294.869} C_VEL
LIN {X 0,Y 277.809,Z 424.879,A -85,B 0,C 180,E1 -18295.159,E2 -18295.159} C_VEL
LIN {X 0,Y 274.249,Z 412.753,A -85,B 0,C 180,E1 -18296.377,E2 -18296.377} C_VEL
LIN {X 0,Y 269.432,Z 399.984,A -85,B 0,C 180,E1 -18297.471,E2 -18297.471} C_VEL
LIN {X 0,Y 269.488,Z 389.375,A -85,B 0,C 180,E1 -18302.313,E2 -18302.313} C_VEL
LIN {X 0,Y 269.816,Z 380.097,A -85,B 0,C 180,E1 -18306.799,E2 -18306.799} C_VEL
LIN {X 0,Y 269.62,Z 376.504,A -85,B 0,C 180,E1 -18308.72,E2 -18308.72} C_VEL
LIN {X 0,Y 268.314,Z 368.982,A -85,B 0,C 180,E1 -18312.826,E2 -18312.826} C_VEL
LIN {X 0,Y 266.872,Z 361.979,A -85,B 0,C 180,E1 -18316.787,E2 -18316.787} C_VEL
LIN {X 0,Y 265.383,Z 355.629,A -85,B 0,C 180,E1 -18320.536,E2 -18320.536} C_VEL
LIN {X 0,Y 263.971,Z 350.737,A -85,B 0,C 180,E1 -18323.446,E2 -18323.446} C_VEL
LIN {X 0,Y 263.178,Z 348.013,A -85,B 0,C 180,E1 -18325.077,E2 -18325.077} C_VEL
LIN {X 0,Y 263.133,Z 348.015,A -85,B 0,C 180,E1 -18329.504,E2 -18329.504} C_VEL
LIN {X 0,Y 263.177,Z 348.006,A -85,B 0,C 180,E1 -18333,E2 -18333} C_VEL
LIN {X 0,Y 263.202,Z 348.004,A -85,B 0,C 180,E1 -18336.388,E2 -18336.388} C_VEL
LIN {X 0,Y 263.273,Z 348.002,A -85,B 0,C 180,E1 -18339.693,E2 -18339.693} C_VEL
LIN {X 0,Y 263.325,Z 347.989,A -85,B 0,C 180,E1 -18344.52,E2 -18344.52} C_VEL
LIN {X 0,Y 263.353,Z 347.986,A -85,B 0,C 180,E1 -18349.233,E2 -18349.233} C_VEL
LIN {X 0,Y 263.55,Z 347.966,A -85,B 0,C 180,E1 -18352.337,E2 -18352.337} C_VEL
LIN {X 0,Y 263.728,Z 347.948,A -85,B 0,C 180,E1 -18358.472,E2 -18358.472} C_VEL
LIN {X 0,Y 263.737,Z 347.931,A -85,B 0,C 180,E1 -18361.526,E2 -18361.526} C_VEL
LIN {X 0,Y 263.551,Z 347.97,A -85,B 0,C 180,E1 -18367.662,E2 -18367.662} C_VEL
LIN {X 0,Y 263.333,Z 347.995,A -85,B 0,C 180,E1 -18371.012,E2 -18371.012} C_VEL
LIN {X 0,Y 262.611,Z 348.088,A -85,B 0,C 180,E1 -18371.861,E2 -18371.861} C_VEL
LIN {X 0,Y 259.73,Z 348.444,A -85,B 0,C 180,E1 -18373.192,E2 -18373.192} C_VEL
LIN {X 0,Y 256.883,Z 348.799,A -85,B 0,C 180,E1 -18374.551,E2 -18374.551} C_VEL
LIN {X 0,Y 256.244,Z 348.878,A -85,B 0,C 180,E1 -18375.432,E2 -18375.432} C_VEL
LIN {X 0,Y 256.198,Z 348.916,A -85,B 0,C 180,E1 -18377.562,E2 -18377.562} C_VEL
LIN {X 0,Y 257.965,Z 355.7,A -85,B 0,C 180,E1 -18382.148,E2 -18382.148} C_VEL
LIN {X 0,Y 259.762,Z 362.591,A -85,B 0,C 180,E1 -18386.386,E2 -18386.386} C_VEL
LIN {X 0,Y 261.38,Z 368.632,A -85,B 0,C 180,E1 -18389.829,E2 -18389.829} C_VEL
LIN {X 0,Y 263.676,Z 377.104,A -85,B 0,C 180,E1 -18394.291,E2 -18394.291} C_VEL
LIN {X 0,Y 265.949,Z 385.582,A -85,B 0,C 180,E1 -18398.389,E2 -18398.389} C_VEL
LIN {X 0,Y 268.383,Z 394.543,A -85,B 0,C 180,E1 -18402.399,E2 -18402.399} C_VEL
LIN {X 0,Y 270.735,Z 402.832,A -85,B 0,C 180,E1 -18405.866,E2 -18405.866} C_VEL
LIN {X 0,Y 272.151,Z 408.99,A -85,B 0,C 180,E1 -18408.277,E2 -18408.277} C_VEL
LIN {X 0,Y 271.695,Z 410.616,A -85,B 0,C 180,E1 -18408.816,E2 -18408.816} C_VEL
LIN {X 0,Y 273.65,Z 430.168,A -85,B 0,C 180,E1 -18409.928,E2 -18409.928} C_VEL
LIN {X 0,Y 275.378,Z 447.488,A -85,B 0,C 180,E1 -18411.197,E2 -18411.197} C_VEL
LIN {X 0,Y 276.891,Z 464.181,A -85,B 0,C 180,E1 -18412.705,E2 -18412.705} C_VEL
LIN {X 0,Y 277.411,Z 473.798,A -85,B 0,C 180,E1 -18413.693,E2 -18413.693} C_VEL
LIN {X 0,Y 274.811,Z 488.011,A -85,B 0,C 180,E1 -18415.138,E2 -18415.138} C_VEL
LIN {X 0,Y 271.777,Z 502.208,A -85,B 0,C 180,E1 -18416.893,E2 -18416.893} C_VEL
LIN {X 0,Y 269,Z 514.436,A -85,B 0,C 180,E1 -18418.722,E2 -18418.722} C_VEL
LIN {X 0,Y 265.956,Z 527.156,A -85,B 0,C 180,E1 -18420.985,E2 -18420.985} C_VEL
LIN {X 0,Y 263.182,Z 538.654,A -85,B 0,C 180,E1 -18423.435,E2 -18423.435} C_VEL
LIN {X 0,Y 260.668,Z 549.312,A -85,B 0,C 180,E1 -18426.15,E2 -18426.15} C_VEL
LIN {X 0,Y 258.699,Z 558.392,A -85,B 0,C 180,E1 -18428.907,E2 -18428.907} C_VEL
LIN {X 0,Y 257.307,Z 566.041,A -85,B 0,C 180,E1 -18431.697,E2 -18431.697} C_VEL
LIN {X 0,Y 256.137,Z 573.26,A -85,B 0,C 180,E1 -18434.895,E2 -18434.895} C_VEL
LIN {X 0,Y 255.514,Z 579.052,A -85,B 0,C 180,E1 -18438.099,E2 -18438.099} C_VEL
LIN {X 0,Y 255.423,Z 582.531,A -85,B 0,C 180,E1 -18440.502,E2 -18440.502} C_VEL
LIN {X 0,Y 255.465,Z 586.03,A -85,B 0,C 180,E1 -18443.686,E2 -18443.686} C_VEL
LIN {X 0,Y 255.578,Z 588.301,A -85,B 0,C 180,E1 -18446.851,E2 -18446.851} C_VEL
LIN {X 0,Y 255.655,Z 589.293,A -85,B 0,C 180,E1 -18450.004,E2 -18450.004} C_VEL
LIN {X 0,Y 255.476,Z 589.136,A -85,B 0,C 180,E1 -18453.158,E2 -18453.158} C_VEL
LIN {X 0,Y 255.457,Z 588.647,A -85,B 0,C 180,E1 -18454.738,E2 -18454.738} C_VEL
LIN {X 0,Y 255.11,Z 586.714,A -85,B 0,C 180,E1 -18457.921,E2 -18457.921} C_VEL
LIN {X 0,Y 255.075,Z 583.81,A -85,B 0,C 180,E1 -18461.124,E2 -18461.124} C_VEL
LIN {X 0,Y 255.775,Z 578.685,A -85,B 0,C 180,E1 -18465.135,E2 -18465.135} C_VEL
LIN {X 0,Y 257.31,Z 571.924,A -85,B 0,C 180,E1 -18469.137,E2 -18469.137} C_VEL
LIN {X 0,Y 260.043,Z 563.16,A -85,B 0,C 180,E1 -18473.237,E2 -18473.237} C_VEL
LIN {X 0,Y 263.75,Z 553.372,A -85,B 0,C 180,E1 -18476.939,E2 -18476.939} C_VEL
LIN {X 0,Y 268.87,Z 541.596,A -85,B 0,C 180,E1 -18480.561,E2 -18480.561} C_VEL
LIN {X 0,Y 273.991,Z 530.264,A -85,B 0,C 180,E1 -18483.472,E2 -18483.472} C_VEL
LIN {X 0,Y 280.757,Z 515.944,A -85,B 0,C 180,E1 -18486.482,E2 -18486.482} C_VEL
LIN {X 0,Y 287.702,Z 501.356,A -85,B 0,C 180,E1 -18488.981,E2 -18488.981} C_VEL
LIN {X 0,Y 295.376,Z 484.634,A -85,B 0,C 180,E1 -18491.323,E2 -18491.323} C_VEL
LIN {X 0,Y 300.019,Z 471.437,A -85,B 0,C 180,E1 -18493.299,E2 -18493.299} C_VEL
LIN {X 0,Y 302.869,Z 462.817,A -85,B 0,C 180,E1 -18494.577,E2 -18494.577} C_VEL
LIN {X 0,Y 305.572,Z 453.442,A -85,B 0,C 180,E1 -18496.184,E2 -18496.184} C_VEL
LIN {X 0,Y 305.618,Z 452.826,A -85,B 0,C 180,E1 -18496.38,E2 -18496.38} C_VEL
LIN {X 0,Y 304.591,Z 450.893,A -85,B 0,C 180,E1 -18498.001,E2 -18498.001} C_VEL
LIN {X 0,Y 303.856,Z 449.58,A -85,B 0,C 180,E1 -18499.757,E2 -18499.757} C_VEL
LIN {X 0,Y 303.36,Z 449.406,A -85,B 0,C 180,E1 -18501.281,E2 -18501.281} C_VEL
LIN {X 0,Y 302.729,Z 450.405,A -85,B 0,C 180,E1 -18502.872,E2 -18502.872} C_VEL
LIN {X 0,Y 301.829,Z 453.596,A -85,B 0,C 180,E1 -18505.185,E2 -18505.185} C_VEL
LIN {X 0,Y 301.116,Z 457.376,A -85,B 0,C 180,E1 -18507.169,E2 -18507.169} C_VEL
LIN {X 0,Y 300.491,Z 460.905,A -85,B 0,C 180,E1 -18508.642,E2 -18508.642} C_VEL
LIN {X 0,Y 293.333,Z 473.675,A -85,B 0,C 180,E1 -18510.977,E2 -18510.977} C_VEL
LIN {X 0,Y 287.687,Z 483.165,A -85,B 0,C 180,E1 -18513.132,E2 -18513.132} C_VEL
LIN {X 0,Y 282.508,Z 491.328,A -85,B 0,C 180,E1 -18515.375,E2 -18515.375} C_VEL
LIN {X 0,Y 277.848,Z 498.229,A -85,B 0,C 180,E1 -18517.703,E2 -18517.703} C_VEL
LIN {X 0,Y 273.148,Z 504.645,A -85,B 0,C 180,E1 -18520.459,E2 -18520.459} C_VEL
LIN {X 0,Y 269.069,Z 509.62,A -85,B 0,C 180,E1 -18523.303,E2 -18523.303} C_VEL
LIN {X 0,Y 265.582,Z 513.196,A -85,B 0,C 180,E1 -18526.222,E2 -18526.222} C_VEL
LIN {X 0,Y 262.835,Z 515.355,A -85,B 0,C 180,E1 -18529.213,E2 -18529.213} C_VEL
LIN {X 0,Y 260.776,Z 516.054,A -85,B 0,C 180,E1 -18532.256,E2 -18532.256} C_VEL
LIN {X 0,Y 259.169,Z 515.308,A -85,B 0,C 180,E1 -18535.334,E2 -18535.334} C_VEL
LIN {X 0,Y 258.423,Z 514.403,A -85,B 0,C 180,E1 -18536.883,E2 -18536.883} C_VEL
LIN {X 0,Y 257.523,Z 511.39,A -85,B 0,C 180,E1 -18540.001,E2 -18540.001} C_VEL
LIN {X 0,Y 257.232,Z 508.042,A -85,B 0,C 180,E1 -18542.349,E2 -18542.349} C_VEL
LIN {X 0,Y 257.241,Z 503.751,A -85,B 0,C 180,E1 -18544.702,E2 -18544.702} C_VEL
LIN {X 0,Y 257.208,Z 498.475,A -85,B 0,C 180,E1 -18547.064,E2 -18547.064} C_VEL
LIN {X 0,Y 258.004,Z 490.85,A -85,B 0,C 180,E1 -18549.803,E2 -18549.803} C_VEL
LIN {X 0,Y 258.746,Z 481.535,A -85,B 0,C 180,E1 -18552.551,E2 -18552.551} C_VEL
LIN {X 0,Y 259.791,Z 471.896,A -85,B 0,C 180,E1 -18554.893,E2 -18554.893} C_VEL
LIN {X 0,Y 261.028,Z 460.449,A -85,B 0,C 180,E1 -18557.228,E2 -18557.228} C_VEL
LIN {X 0,Y 262.637,Z 447.904,A -85,B 0,C 180,E1 -18559.339,E2 -18559.339} C_VEL
LIN {X 0,Y 264.275,Z 432.758,A -85,B 0,C 180,E1 -18561.438,E2 -18561.438} C_VEL
LIN {X 0,Y 265.729,Z 419.221,A -85,B 0,C 180,E1 -18562.962,E2 -18562.962} C_VEL
LIN {X 0,Y 265.772,Z 415.369,A -85,B 0,C 180,E1 -18563.37,E2 -18563.37} C_VEL
LIN {X 0,Y 262.746,Z 399.945,A -85,B 0,C 180,E1 -18565.022,E2 -18565.022} C_VEL
LIN {X 0,Y 258.993,Z 383.874,A -85,B 0,C 180,E1 -18566.502,E2 -18566.502} C_VEL
LIN {X 0,Y 257.235,Z 376.603,A -85,B 0,C 180,E1 -18567.119,E2 -18567.119} C_VEL
LIN {X 0,Y 257.78,Z 370.783,A -85,B 0,C 180,E1 -18571.199,E2 -18571.199} C_VEL
LIN {X 0,Y 258.333,Z 365.16,A -85,B 0,C 180,E1 -18575.293,E2 -18575.293} C_VEL
LIN {X 0,Y 258.224,Z 360.658,A -85,B 0,C 180,E1 -18578.755,E2 -18578.755} C_VEL
LIN {X 0,Y 258.015,Z 359.441,A -85,B 0,C 180,E1 -18579.748,E2 -18579.748} C_VEL
LIN {X 0,Y 259.947,Z 363.734,A -85,B 0,C 180,E1 -18582.525,E2 -18582.525} C_VEL
LIN {X 0,Y 260.797,Z 366.902,A -85,B 0,C 180,E1 -18584.48,E2 -18584.48} C_VEL
LIN {X 0,Y 262.344,Z 374.801,A -85,B 0,C 180,E1 -18588.985,E2 -18588.985} C_VEL
LIN {X 0,Y 263.166,Z 380.434,A -85,B 0,C 180,E1 -18592.1,E2 -18592.1} C_VEL
LIN {X 0,Y 262.926,Z 388.192,A -85,B 0,C 180,E1 -18595.959,E2 -18595.959} C_VEL
LIN {X 0,Y 262.68,Z 397.486,A -85,B 0,C 180,E1 -18600.329,E2 -18600.329} C_VEL
LIN {X 0,Y 262.731,Z 400.98,A -85,B 0,C 180,E1 -18601.89,E2 -18601.89} C_VEL
LIN {X 0,Y 267.609,Z 413.723,A -85,B 0,C 180,E1 -18603.036,E2 -18603.036} C_VEL
LIN {X 0,Y 271.132,Z 425.49,A -85,B 0,C 180,E1 -18604.26,E2 -18604.26} C_VEL
LIN {X 0,Y 271.574,Z 428.273,A -85,B 0,C 180,E1 -18604.548,E2 -18604.548} C_VEL
LIN {X 0,Y 270.457,Z 439.871,A -85,B 0,C 180,E1 -18605.611,E2 -18605.611} C_VEL
LIN {X 0,Y 268.954,Z 450.9,A -85,B 0,C 180,E1 -18606.92,E2 -18606.92} C_VEL
LIN {X 0,Y 267.269,Z 461.921,A -85,B 0,C 180,E1 -18608.598,E2 -18608.598} C_VEL
LIN {X 0,Y 266.042,Z 468.945,A -85,B 0,C 180,E1 -18609.911,E2 -18609.911} C_VEL
LIN {X 0,Y 264.336,Z 477.408,A -85,B 0,C 180,E1 -18611.792,E2 -18611.792} C_VEL
LIN {X 0,Y 262.494,Z 485.633,A -85,B 0,C 180,E1 -18614.068,E2 -18614.068} C_VEL
LIN {X 0,Y 261.355,Z 491.187,A -85,B 0,C 180,E1 -18615.991,E2 -18615.991} C_VEL
LIN {X 0,Y 259.905,Z 496.623,A -85,B 0,C 180,E1 -18618.295,E2 -18618.295} C_VEL
LIN {X 0,Y 258.581,Z 500.906,A -85,B 0,C 180,E1 -18620.611,E2 -18620.611} C_VEL
LIN {X 0,Y 258.074,Z 503.126,A -85,B 0,C 180,E1 -18622.171,E2 -18622.171} C_VEL
LIN {X 0,Y 257.814,Z 504.913,A -85,B 0,C 180,E1 -18623.736,E2 -18623.736} C_VEL
LIN {X 0,Y 257.438,Z 506.301,A -85,B 0,C 180,E1 -18625.299,E2 -18625.299} C_VEL
LIN {X 0,Y 257.072,Z 507.864,A -85,B 0,C 180,E1 -18628.43,E2 -18628.43} C_VEL
LIN {X 0,Y 257.023,Z 508.092,A -85,B 0,C 180,E1 -18629.996,E2 -18629.996} C_VEL
LIN {X 0,Y 257.162,Z 507.336,A -85,B 0,C 180,E1 -18633.129,E2 -18633.129} C_VEL
LIN {X 0,Y 257.814,Z 505.046,A -85,B 0,C 180,E1 -18636.256,E2 -18636.256} C_VEL
LIN {X 0,Y 258.337,Z 502.266,A -85,B 0,C 180,E1 -18638.601,E2 -18638.601} C_VEL
LIN {X 0,Y 259.409,Z 498.427,A -85,B 0,C 180,E1 -18640.928,E2 -18640.928} C_VEL
LIN {X 0,Y 260.827,Z 493.434,A -85,B 0,C 180,E1 -18643.236,E2 -18643.236} C_VEL
LIN {X 0,Y 262.207,Z 487.183,A -85,B 0,C 180,E1 -18645.543,E2 -18645.543} C_VEL
LIN {X 0,Y 263.96,Z 479.378,A -85,B 0,C 180,E1 -18647.825,E2 -18647.825} C_VEL
LIN {X 0,Y 265.612,Z 471.381,A -85,B 0,C 180,E1 -18649.712,E2 -18649.712} C_VEL
LIN {X 0,Y 267.193,Z 462.64,A -85,B 0,C 180,E1 -18651.4,E2 -18651.4} C_VEL
LIN {X 0,Y 268.856,Z 451.778,A -85,B 0,C 180,E1 -18653.081,E2 -18653.081} C_VEL
LIN {X 0,Y 270.354,Z 441.135,A -85,B 0,C 180,E1 -18654.369,E2 -18654.369} C_VEL
LIN {X 0,Y 271.5,Z 429.933,A -85,B 0,C 180,E1 -18655.435,E2 -18655.435} C_VEL
LIN {X 0,Y 271.647,Z 428.043,A -85,B 0,C 180,E1 -18655.587,E2 -18655.587} C_VEL
LIN {X 0,Y 269.062,Z 418.209,A -85,B 0,C 180,E1 -18656.643,E2 -18656.643} C_VEL
LIN {X 0,Y 264.951,Z 406.581,A -85,B 0,C 180,E1 -18657.743,E2 -18657.743} C_VEL
LIN {X 0,Y 262.779,Z 401.033,A -85,B 0,C 180,E1 -18658.231,E2 -18658.231} C_VEL
LIN {X 0,Y 262.836,Z 392.071,A -85,B 0,C 180,E1 -18662.324,E2 -18662.324} C_VEL
LIN {X 0,Y 263.219,Z 383.025,A -85,B 0,C 180,E1 -18666.773,E2 -18666.773} C_VEL
LIN {X 0,Y 262.921,Z 378.447,A -85,B 0,C 180,E1 -18669.177,E2 -18669.177} C_VEL
LIN {X 0,Y 261.88,Z 372.485,A -85,B 0,C 180,E1 -18672.454,E2 -18672.454} C_VEL
LIN {X 0,Y 260.428,Z 364.989,A -85,B 0,C 180,E1 -18676.765,E2 -18676.765} C_VEL
LIN {X 0,Y 259.049,Z 359.038,A -85,B 0,C 180,E1 -18680.389,E2 -18680.389} C_VEL
LIN {X 0,Y 257.833,Z 354.534,A -85,B 0,C 180,E1 -18683.153,E2 -18683.153} C_VEL
LIN {X 0,Y 256.069,Z 348.895,A -85,B 0,C 180,E1 -18686.707,E2 -18686.707} C_VEL
LIN {X 0,Y 256.121,Z 348.894,A -85,B 0,C 180,E1 -18691.402,E2 -18691.402} C_VEL
LIN {X 0,Y 256.169,Z 348.887,A -85,B 0,C 180,E1 -18695.699,E2 -18695.699} C_VEL
LIN {X 0,Y 256.222,Z 348.883,A -85,B 0,C 180,E1 -18699.109,E2 -18699.109} C_VEL
LIN {X 0,Y 256.275,Z 348.873,A -85,B 0,C 180,E1 -18704.083,E2 -18704.083} C_VEL
LIN {X 0,Y 256.289,Z 348.869,A -85,B 0,C 180,E1 -18708.932,E2 -18708.932} C_VEL
LIN {X 0,Y 256.518,Z 348.839,A -85,B 0,C 180,E1 -18712.126,E2 -18712.126} C_VEL
LIN {X 0,Y 256.691,Z 348.825,A -85,B 0,C 180,E1 -18718.43,E2 -18718.43} C_VEL
LIN {X 0,Y 256.701,Z 348.807,A -85,B 0,C 180,E1 -18721.568,E2 -18721.568} C_VEL
LIN {X 0,Y 256.518,Z 348.847,A -85,B 0,C 180,E1 -18727.873,E2 -18727.873} C_VEL
LIN {X 0,Y 256.288,Z 348.873,A -85,B 0,C 180,E1 -18731.066,E2 -18731.066} C_VEL
LIN {X 0,Y 256.244,Z 348.878,A -85,B 0,C 180,E1 -18735.432,E2 -18735.432} C_VEL
LIN {X 0,Y 256.025,Z 349.153,A -85,B 0,C 180,E1 -18736.305,E2 -18736.305} C_VEL
LIN {X 0,Y 255.399,Z 349.888,A -85,B 0,C 180,E1 -18737.158,E2 -18737.158} C_VEL
LIN {X 0,Y 253.539,Z 352.29,A -85,B 0,C 180,E1 -18738.81,E2 -18738.81} C_VEL
LIN {X 0,Y 251.788,Z 355.356,A -85,B 0,C 180,E1 -18740.46,E2 -18740.46} C_VEL
LIN {X 0,Y 251.274,Z 357.636,A -85,B 0,C 180,E1 -18741.726,E2 -18741.726} C_VEL
LIN {X 0,Y 251.36,Z 358.328,A -85,B 0,C 180,E1 -18742.156,E2 -18742.156} C_VEL
LIN {X 0,Y 253.126,Z 365.066,A -85,B 0,C 180,E1 -18746.374,E2 -18746.374} C_VEL
LIN {X 0,Y 255.053,Z 372.49,A -85,B 0,C 180,E1 -18750.634,E2 -18750.634} C_VEL
LIN {X 0,Y 257.325,Z 380.741,A -85,B 0,C 180,E1 -18754.997,E2 -18754.997} C_VEL
LIN {X 0,Y 259.818,Z 389.971,A -85,B 0,C 180,E1 -18759.469,E2 -18759.469} C_VEL
LIN {X 0,Y 262.643,Z 400.336,A -85,B 0,C 180,E1 -18764.084,E2 -18764.084} C_VEL
LIN {X 0,Y 264.848,Z 408.409,A -85,B 0,C 180,E1 -18767.43,E2 -18767.43} C_VEL
LIN {X 0,Y 265.152,Z 410.284,A -85,B 0,C 180,E1 -18768.138,E2 -18768.138} C_VEL
LIN {X 0,Y 267.025,Z 430.36,A -85,B 0,C 180,E1 -18769.324,E2 -18769.324} C_VEL
LIN {X 0,Y 268.603,Z 447.192,A -85,B 0,C 180,E1 -18770.593,E2 -18770.593} C_VEL
LIN {X 0,Y 270.104,Z 463.549,A -85,B 0,C 180,E1 -18772.114,E2 -18772.114} C_VEL
LIN {X 0,Y 270.584,Z 474.899,A -85,B 0,C 180,E1 -18773.322,E2 -18773.322} C_VEL
LIN {X 0,Y 267.58,Z 489.949,A -85,B 0,C 180,E1 -18774.937,E2 -18774.937} C_VEL
LIN {X 0,Y 264.222,Z 505.179,A -85,B 0,C 180,E1 -18776.962,E2 -18776.962} C_VEL
LIN {X 0,Y 261.131,Z 517.971,A -85,B 0,C 180,E1 -18779.026,E2 -18779.026} C_VEL
LIN {X 0,Y 258.439,Z 529.038,A -85,B 0,C 180,E1 -18781.144,E2 -18781.144} C_VEL
LIN {X 0,Y 255.489,Z 541.022,A -85,B 0,C 180,E1 -18783.893,E2 -18783.893} C_VEL
LIN {X 0,Y 252.983,Z 551.483,A -85,B 0,C 180,E1 -18786.796,E2 -18786.796} C_VEL
LIN {X 0,Y 250.992,Z 560.86,A -85,B 0,C 180,E1 -18789.944,E2 -18789.944} C_VEL
LIN {X 0,Y 249.785,Z 567.849,A -85,B 0,C 180,E1 -18792.774,E2 -18792.774} C_VEL
LIN {X 0,Y 248.825,Z 574.613,A -85,B 0,C 180,E1 -18796.113,E2 -18796.113} C_VEL
LIN {X 0,Y 248.427,Z 579.899,A -85,B 0,C 180,E1 -18799.408,E2 -18799.408} C_VEL
LIN {X 0,Y 248.422,Z 583.03,A -85,B 0,C 180,E1 -18801.955,E2 -18801.955} C_VEL
LIN {X 0,Y 248.513,Z 585.942,A -85,B 0,C 180,E1 -18805.137,E2 -18805.137} C_VEL
LIN {X 0,Y 248.653,Z 587.633,A -85,B 0,C 180,E1 -18808.384,E2 -18808.384} C_VEL
LIN {X 0,Y 248.676,Z 588.041,A -85,B 0,C 180,E1 -18810.004,E2 -18810.004} C_VEL
LIN {X 0,Y 248.459,Z 587.977,A -85,B 0,C 180,E1 -18813.247,E2 -18813.247} C_VEL
LIN {X 0,Y 248.422,Z 587.479,A -85,B 0,C 180,E1 -18814.872,E2 -18814.872} C_VEL
LIN {X 0,Y 248.047,Z 585.656,A -85,B 0,C 180,E1 -18818.148,E2 -18818.148} C_VEL
LIN {X 0,Y 248.019,Z 582.81,A -85,B 0,C 180,E1 -18821.445,E2 -18821.445} C_VEL
LIN {X 0,Y 248.563,Z 578.926,A -85,B 0,C 180,E1 -18824.746,E2 -18824.746} C_VEL
LIN {X 0,Y 249.653,Z 574.069,A -85,B 0,C 180,E1 -18828.043,E2 -18828.043} C_VEL
LIN {X 0,Y 251.988,Z 566.519,A -85,B 0,C 180,E1 -18832.122,E2 -18832.122} C_VEL
LIN {X 0,Y 255.55,Z 557.346,A -85,B 0,C 180,E1 -18836.109,E2 -18836.109} C_VEL
LIN {X 0,Y 260.43,Z 546.57,A -85,B 0,C 180,E1 -18839.909,E2 -18839.909} C_VEL
LIN {X 0,Y 266.015,Z 535.034,A -85,B 0,C 180,E1 -18843.248,E2 -18843.248} C_VEL
LIN {X 0,Y 272.671,Z 521.95,A -85,B 0,C 180,E1 -18846.361,E2 -18846.361} C_VEL
LIN {X 0,Y 279.586,Z 508.684,A -85,B 0,C 180,E1 -18848.938,E2 -18848.938} C_VEL
LIN {X 0,Y 286.369,Z 495.541,A -85,B 0,C 180,E1 -18851.036,E2 -18851.036} C_VEL
LIN {X 0,Y 290.467,Z 487.376,A -85,B 0,C 180,E1 -18852.18,E2 -18852.18} C_VEL
LIN {X 0,Y 298.494,Z 467.154,A -85,B 0,C 180,E1 -18855.319,E2 -18855.319} C_VEL
LIN {X 0,Y 301.44,Z 458.761,A -85,B 0,C 180,E1 -18856.796,E2 -18856.796} C_VEL
LIN {X 0,Y 301.251,Z 457.668,A -85,B 0,C 180,E1 -18857.426,E2 -18857.426} C_VEL
LIN {X 0,Y 300.441,Z 456.131,A -85,B 0,C 180,E1 -18859.082,E2 -18859.082} C_VEL
LIN {X 0,Y 299.81,Z 455.518,A -85,B 0,C 180,E1 -18860.735,E2 -18860.735} C_VEL
LIN {X 0,Y 299.126,Z 456.111,A -85,B 0,C 180,E1 -18862.348,E2 -18862.348} C_VEL
LIN {X 0,Y 297.896,Z 458.88,A -85,B 0,C 180,E1 -18864.657,E2 -18864.657} C_VEL
LIN {X 0,Y 297.103,Z 461.494,A -85,B 0,C 180,E1 -18866.227,E2 -18866.227} C_VEL
LIN {X 0,Y 296.201,Z 464.7,A -85,B 0,C 180,E1 -18867.733,E2 -18867.733} C_VEL
LIN {X 0,Y 294.482,Z 467.82,A -85,B 0,C 180,E1 -18868.329,E2 -18868.329} C_VEL
LIN {X 0,Y 287.993,Z 478.198,A -85,B 0,C 180,E1 -18870.386,E2 -18870.386} C_VEL
LIN {X 0,Y 281.229,Z 488.309,A -85,B 0,C 180,E1 -18872.867,E2 -18872.867} C_VEL
LIN {X 0,Y 275.929,Z 495.766,A -85,B 0,C 180,E1 -18875.15,E2 -18875.15} C_VEL
LIN {X 0,Y 270.541,Z 502.889,A -85,B 0,C 180,E1 -18877.873,E2 -18877.873} C_VEL
LIN {X 0,Y 265.812,Z 508.541,A -85,B 0,C 180,E1 -18880.702,E2 -18880.702} C_VEL
LIN {X 0,Y 262.647,Z 511.899,A -85,B 0,C 180,E1 -18882.883,E2 -18882.883} C_VEL
LIN {X 0,Y 258.99,Z 515.2,A -85,B 0,C 180,E1 -18885.865,E2 -18885.865} C_VEL
LIN {X 0,Y 256.078,Z 517.054,A -85,B 0,C 180,E1 -18888.924,E2 -18888.924} C_VEL
LIN {X 0,Y 253.889,Z 517.491,A -85,B 0,C 180,E1 -18892.045,E2 -18892.045} C_VEL
LIN {X 0,Y 252.201,Z 516.543,A -85,B 0,C 180,E1 -18895.205,E2 -18895.205} C_VEL
LIN {X 0,Y 250.904,Z 514.11,A -85,B 0,C 180,E1 -18898.396,E2 -18898.396} C_VEL
LIN {X 0,Y 250.34,Z 511.22,A -85,B 0,C 180,E1 -18900.805,E2 -18900.805} C_VEL
LIN {X 0,Y 250.133,Z 507.414,A -85,B 0,C 180,E1 -18903.222,E2 -18903.222} C_VEL
LIN {X 0,Y 250.142,Z 502.643,A -85,B 0,C 180,E1 -18905.644,E2 -18905.644} C_VEL
LIN {X 0,Y 250.451,Z 495.726,A -85,B 0,C 180,E1 -18908.472,E2 -18908.472} C_VEL
LIN {X 0,Y 251.148,Z 488.541,A -85,B 0,C 180,E1 -18910.889,E2 -18910.889} C_VEL
LIN {X 0,Y 252.128,Z 478.44,A -85,B 0,C 180,E1 -18913.706,E2 -18913.706} C_VEL
LIN {X 0,Y 253.325,Z 467.99,A -85,B 0,C 180,E1 -18916.108,E2 -18916.108} C_VEL
LIN {X 0,Y 254.79,Z 455.578,A -85,B 0,C 180,E1 -18918.495,E2 -18918.495} C_VEL
LIN {X 0,Y 256.454,Z 441.903,A -85,B 0,C 180,E1 -18920.661,E2 -18920.661} C_VEL
LIN {X 0,Y 258.085,Z 426.77,A -85,B 0,C 180,E1 -18922.622,E2 -18922.622} C_VEL
LIN {X 0,Y 259.081,Z 417.797,A -85,B 0,C 180,E1 -18923.586,E2 -18923.586} C_VEL
LIN {X 0,Y 256.396,Z 403.289,A -85,B 0,C 180,E1 -18925.231,E2 -18925.231} C_VEL
LIN {X 0,Y 252.604,Z 386.521,A -85,B 0,C 180,E1 -18926.862,E2 -18926.862} C_VEL
LIN {X 0,Y 250.313,Z 377.015,A -85,B 0,C 180,E1 -18927.695,E2 -18927.695} C_VEL
LIN {X 0,Y 250.796,Z 372.068,A -85,B 0,C 180,E1 -18931.227,E2 -18931.227} C_VEL
LIN {X 0,Y 251.313,Z 367.064,A -85,B 0,C 180,E1 -18934.911,E2 -18934.911} C_VEL
LIN {X 0,Y 251.28,Z 362.515,A -85,B 0,C 180,E1 -18938.448,E2 -18938.448} C_VEL
LIN {X 0,Y 251.238,Z 361.812,A -85,B 0,C 180,E1 -18939.098,E2 -18939.098} C_VEL
LIN {X 0,Y 253.109,Z 365.684,A -85,B 0,C 180,E1 -18941.791,E2 -18941.791} C_VEL
LIN {X 0,Y 254.238,Z 369.239,A -85,B 0,C 180,E1 -18944.046,E2 -18944.046} C_VEL
LIN {X 0,Y 255.536,Z 375.903,A -85,B 0,C 180,E1 -18947.953,E2 -18947.953} C_VEL
LIN {X 0,Y 256.371,Z 381.125,A -85,B 0,C 180,E1 -18950.908,E2 -18950.908} C_VEL
LIN {X 0,Y 256.527,Z 384.938,A -85,B 0,C 180,E1 -18952.931,E2 -18952.931} C_VEL
LIN {X 0,Y 256.231,Z 392.648,A -85,B 0,C 180,E1 -18956.727,E2 -18956.727} C_VEL
LIN {X 0,Y 256.115,Z 402.18,A -85,B 0,C 180,E1 -18961.128,E2 -18961.128} C_VEL
LIN {X 0,Y 261.008,Z 414.669,A -85,B 0,C 180,E1 -18962.289,E2 -18962.289} C_VEL
LIN {X 0,Y 264.234,Z 425.375,A -85,B 0,C 180,E1 -18963.427,E2 -18963.427} C_VEL
LIN {X 0,Y 265.218,Z 429.641,A -85,B 0,C 180,E1 -18963.919,E2 -18963.919} C_VEL
LIN {X 0,Y 264.073,Z 440.927,A -85,B 0,C 180,E1 -18964.981,E2 -18964.981} C_VEL
LIN {X 0,Y 262.511,Z 451.966,A -85,B 0,C 180,E1 -18966.319,E2 -18966.319} C_VEL
LIN {X 0,Y 260.744,Z 462.992,A -85,B 0,C 180,E1 -18968.035,E2 -18968.035} C_VEL
LIN {X 0,Y 259.461,Z 470.018,A -85,B 0,C 180,E1 -18969.379,E2 -18969.379} C_VEL
LIN {X 0,Y 257.678,Z 478.482,A -85,B 0,C 180,E1 -18971.305,E2 -18971.305} C_VEL
LIN {X 0,Y 255.762,Z 486.707,A -85,B 0,C 180,E1 -18973.637,E2 -18973.637} C_VEL
LIN {X 0,Y 254.562,Z 492.262,A -85,B 0,C 180,E1 -18975.609,E2 -18975.609} C_VEL
LIN {X 0,Y 253.038,Z 497.7,A -85,B 0,C 180,E1 -18977.973,E2 -18977.973} C_VEL
LIN {X 0,Y 251.661,Z 501.983,A -85,B 0,C 180,E1 -18980.35,E2 -18980.35} C_VEL
LIN {X 0,Y 251.123,Z 504.204,A -85,B 0,C 180,E1 -18981.952,E2 -18981.952} C_VEL
LIN {X 0,Y 250.837,Z 505.99,A -85,B 0,C 180,E1 -18983.561,E2 -18983.561} C_VEL
LIN {X 0,Y 250.445,Z 507.378,A -85,B 0,C 180,E1 -18985.167,E2 -18985.167} C_VEL
LIN {X 0,Y 250.071,Z 508.939,A -85,B 0,C 180,E1 -18988.386,E2 -18988.386} C_VEL
LIN {X 0,Y 250.018,Z 509.167,A -85,B 0,C 180,E1 -18989.996,E2 -18989.996} C_VEL
LIN {X 0,Y 250.166,Z 508.411,A -85,B 0,C 180,E1 -18993.217,E2 -18993.217} C_VEL
LIN {X 0,Y 250.835,Z 506.122,A -85,B 0,C 180,E1 -18996.431,E2 -18996.431} C_VEL
LIN {X 0,Y 251.398,Z 503.342,A -85,B 0,C 180,E1 -18998.841,E2 -18998.841} C_VEL
LIN {X 0,Y 252.523,Z 499.501,A -85,B 0,C 180,E1 -19001.23,E2 -19001.23} C_VEL
LIN {X 0,Y 254.007,Z 494.506,A -85,B 0,C 180,E1 -19003.598,E2 -19003.598} C_VEL
LIN {X 0,Y 255.452,Z 488.254,A -85,B 0,C 180,E1 -19005.965,E2 -19005.965} C_VEL
LIN {X 0,Y 257.291,Z 480.446,A -85,B 0,C 180,E1 -19008.304,E2 -19008.304} C_VEL
LIN {X 0,Y 259.032,Z 472.445,A -85,B 0,C 180,E1 -19010.234,E2 -19010.234} C_VEL
LIN {X 0,Y 260.671,Z 463.702,A -85,B 0,C 180,E1 -19011.963,E2 -19011.963} C_VEL
LIN {X 0,Y 262.412,Z 452.835,A -85,B 0,C 180,E1 -19013.682,E2 -19013.682} C_VEL
LIN {X 0,Y 263.985,Z 442.109,A -85,B 0,C 180,E1 -19015.006,E2 -19015.006} C_VEL
LIN {X 0,Y 265.151,Z 431.301,A -85,B 0,C 180,E1 -19016.057,E2 -19016.057} C_VEL
LIN {X 0,Y 265.271,Z 429.366,A -85,B 0,C 180,E1 -19016.224,E2 -19016.224} C_VEL
LIN {X 0,Y 261.882,Z 417.275,A -85,B 0,C 180,E1 -19017.569,E2 -19017.569} C_VEL
LIN {X 0,Y 257.301,Z 404.98,A -85,B 0,C 180,E1 -19018.756,E2 -19018.756} C_VEL
LIN {X 0,Y 256.123,Z 402.03,A -85,B 0,C 180,E1 -19019.047,E2 -19019.047} C_VEL
LIN {X 0,Y 256.262,Z 392.964,A -85,B 0,C 180,E1 -19023.259,E2 -19023.259} C_VEL
LIN {X 0,Y 256.631,Z 384.587,A -85,B 0,C 180,E1 -19027.421,E2 -19027.421} C_VEL
LIN {X 0,Y 256.042,Z 379.127,A -85,B 0,C 180,E1 -19030.349,E2 -19030.349} C_VEL
LIN {X 0,Y 254.871,Z 372.465,A -85,B 0,C 180,E1 -19034.197,E2 -19034.197} C_VEL
LIN {X 0,Y 253.857,Z 367.286,A -85,B 0,C 180,E1 -19037.29,E2 -19037.29} C_VEL
LIN {X 0,Y 252.735,Z 362.433,A -85,B 0,C 180,E1 -19040.239,E2 -19040.239} C_VEL
LIN {X 0,Y 251.551,Z 357.951,A -85,B 0,C 180,E1 -19043.08,E2 -19043.08} C_VEL
LIN {X 0,Y 249.87,Z 352.333,A -85,B 0,C 180,E1 -19046.737,E2 -19046.737} C_VEL
LIN {X 0,Y 249.026,Z 349.781,A -85,B 0,C 180,E1 -19048.459,E2 -19048.459} C_VEL
LIN {X 0,Y 249.08,Z 349.77,A -85,B 0,C 180,E1 -19051.335,E2 -19051.335} C_VEL
LIN {X 0,Y 249.143,Z 349.763,A -85,B 0,C 180,E1 -19054.967,E2 -19054.967} C_VEL
LIN {X 0,Y 249.141,Z 349.76,A -85,B 0,C 180,E1 -19058.561,E2 -19058.561} C_VEL
LIN {X 0,Y 249.222,Z 349.754,A -85,B 0,C 180,E1 -19063.62,E2 -19063.62} C_VEL
LIN {X 0,Y 249.232,Z 349.751,A -85,B 0,C 180,E1 -19068.615,E2 -19068.615} C_VEL
LIN {X 0,Y 249.46,Z 349.716,A -85,B 0,C 180,E1 -19071.901,E2 -19071.901} C_VEL
LIN {X 0,Y 249.411,Z 349.719,A -85,B 0,C 180,E1 -19076.769,E2 -19076.769} C_VEL
LIN {X 0,Y 249.699,Z 349.678,A -85,B 0,C 180,E1 -19079.999,E2 -19079.999} C_VEL
LIN {X 0,Y 249.45,Z 349.726,A -85,B 0,C 180,E1 -19083.23,E2 -19083.23} C_VEL
LIN {X 0,Y 249.46,Z 349.725,A -85,B 0,C 180,E1 -19088.097,E2 -19088.097} C_VEL
LIN {X 0,Y 249.231,Z 349.752,A -85,B 0,C 180,E1 -19091.384,E2 -19091.384} C_VEL
LIN {X 0,Y 249.24,Z 349.841,A -85,B 0,C 180,E1 -19096.28,E2 -19096.28} C_VEL
LIN {X 0,Y 251.075,Z 357.065,A -85,B 0,C 180,E1 -19101.339,E2 -19101.339} C_VEL
LIN {X 0,Y 251.36,Z 358.328,A -85,B 0,C 180,E1 -19102.156,E2 -19102.156} C_VEL
LIN {X 0,Y 251.222,Z 360.525,A -85,B 0,C 180,E1 -19103.405,E2 -19103.405} C_VEL
LIN {X 0,Y 249.349,Z 364.76,A -85,B 0,C 180,E1 -19105.414,E2 -19105.414} C_VEL
LIN {X 0,Y 247.531,Z 369.091,A -85,B 0,C 180,E1 -19107.449,E2 -19107.449} C_VEL
LIN {X 0,Y 247.516,Z 371.437,A -85,B 0,C 180,E1 -19108.717,E2 -19108.717} C_VEL
LIN {X 0,Y 249.672,Z 379.661,A -85,B 0,C 180,E1 -19113.291,E2 -19113.291} C_VEL
LIN {X 0,Y 251.548,Z 386.705,A -85,B 0,C 180,E1 -19116.918,E2 -19116.918} C_VEL
LIN {X 0,Y 253.921,Z 395.439,A -85,B 0,C 180,E1 -19121.097,E2 -19121.097} C_VEL
LIN {X 0,Y 256.66,Z 405.119,A -85,B 0,C 180,E1 -19125.393,E2 -19125.393} C_VEL
LIN {X 0,Y 257.89,Z 409.843,A -85,B 0,C 180,E1 -19127.374,E2 -19127.374} C_VEL
LIN {X 0,Y 258.851,Z 413.343,A -85,B 0,C 180,E1 -19127.646,E2 -19127.646} C_VEL
LIN {X 0,Y 260.592,Z 432.614,A -85,B 0,C 180,E1 -19128.853,E2 -19128.853} C_VEL
LIN {X 0,Y 262.141,Z 450.215,A -85,B 0,C 180,E1 -19130.273,E2 -19130.273} C_VEL
LIN {X 0,Y 263.432,Z 466.434,A -85,B 0,C 180,E1 -19131.889,E2 -19131.889} C_VEL
LIN {X 0,Y 263.748,Z 475.649,A -85,B 0,C 180,E1 -19132.914,E2 -19132.914} C_VEL
LIN {X 0,Y 260.657,Z 490.469,A -85,B 0,C 180,E1 -19134.576,E2 -19134.576} C_VEL
LIN {X 0,Y 257.256,Z 505.446,A -85,B 0,C 180,E1 -19136.652,E2 -19136.652} C_VEL
LIN {X 0,Y 254.21,Z 517.585,A -85,B 0,C 180,E1 -19138.685,E2 -19138.685} C_VEL
LIN {X 0,Y 251.142,Z 529.832,A -85,B 0,C 180,E1 -19141.142,E2 -19141.142} C_VEL
LIN {X 0,Y 248.206,Z 541.537,A -85,B 0,C 180,E1 -19143.972,E2 -19143.972} C_VEL
LIN {X 0,Y 245.824,Z 551.468,A -85,B 0,C 180,E1 -19146.857,E2 -19146.857} C_VEL
LIN {X 0,Y 243.804,Z 560.966,A -85,B 0,C 180,E1 -19150.206,E2 -19150.206} C_VEL
LIN {X 0,Y 242.576,Z 567.829,A -85,B 0,C 180,E1 -19153.163,E2 -19153.163} C_VEL
LIN {X 0,Y 241.74,Z 574.282,A -85,B 0,C 180,E1 -19156.555,E2 -19156.555} C_VEL
LIN {X 0,Y 241.433,Z 579.362,A -85,B 0,C 180,E1 -19159.946,E2 -19159.946} C_VEL
LIN {X 0,Y 241.482,Z 583.128,A -85,B 0,C 180,E1 -19163.319,E2 -19163.319} C_VEL
LIN {X 0,Y 241.596,Z 585.539,A -85,B 0,C 180,E1 -19166.669,E2 -19166.669} C_VEL
LIN {X 0,Y 241.693,Z 586.769,A -85,B 0,C 180,E1 -19170.004,E2 -19170.004} C_VEL
LIN {X 0,Y 241.451,Z 586.751,A -85,B 0,C 180,E1 -19173.341,E2 -19173.341} C_VEL
LIN {X 0,Y 241.388,Z 586.307,A -85,B 0,C 180,E1 -19175.015,E2 -19175.015} C_VEL
LIN {X 0,Y 240.983,Z 584.598,A -85,B 0,C 180,E1 -19178.389,E2 -19178.389} C_VEL
LIN {X 0,Y 240.982,Z 581.806,A -85,B 0,C 180,E1 -19181.784,E2 -19181.784} C_VEL
LIN {X 0,Y 241.586,Z 578.073,A -85,B 0,C 180,E1 -19185.182,E2 -19185.182} C_VEL
LIN {X 0,Y 243.175,Z 571.989,A -85,B 0,C 180,E1 -19189.416,E2 -19189.416} C_VEL
LIN {X 0,Y 245.935,Z 564.355,A -85,B 0,C 180,E1 -19193.587,E2 -19193.587} C_VEL
LIN {X 0,Y 249.987,Z 555.128,A -85,B 0,C 180,E1 -19197.641,E2 -19197.641} C_VEL
LIN {X 0,Y 255.504,Z 544.228,A -85,B 0,C 180,E1 -19201.512,E2 -19201.512} C_VEL
LIN {X 0,Y 261.564,Z 532.91,A -85,B 0,C 180,E1 -19204.822,E2 -19204.822} C_VEL
LIN {X 0,Y 268.792,Z 519.963,A -85,B 0,C 180,E1 -19207.915,E2 -19207.915} C_VEL
LIN {X 0,Y 277.157,Z 505.141,A -85,B 0,C 180,E1 -19210.768,E2 -19210.768} C_VEL
LIN {X 0,Y 286.433,Z 488.204,A -85,B 0,C 180,E1 -19213.398,E2 -19213.398} C_VEL
LIN {X 0,Y 294.964,Z 469.461,A -85,B 0,C 180,E1 -19216.44,E2 -19216.44} C_VEL
LIN {X 0,Y 296.79,Z 465.016,A -85,B 0,C 180,E1 -19217.233,E2 -19217.233} C_VEL
LIN {X 0,Y 297.206,Z 463.291,A -85,B 0,C 180,E1 -19217.801,E2 -19217.801} C_VEL
LIN {X 0,Y 296.502,Z 461.99,A -85,B 0,C 180,E1 -19219.335,E2 -19219.335} C_VEL
LIN {X 0,Y 296.141,Z 461.658,A -85,B 0,C 180,E1 -19220.152,E2 -19220.152} C_VEL
LIN {X 0,Y 295.38,Z 461.829,A -85,B 0,C 180,E1 -19221.785,E2 -19221.785} C_VEL
LIN {X 0,Y 294.407,Z 463.154,A -85,B 0,C 180,E1 -19223.36,E2 -19223.36} C_VEL
LIN {X 0,Y 292.917,Z 466.51,A -85,B 0,C 180,E1 -19225.678,E2 -19225.678} C_VEL
LIN {X 0,Y 292.045,Z 468.81,A -85,B 0,C 180,E1 -19226.851,E2 -19226.851} C_VEL
LIN {X 0,Y 290.255,Z 471.61,A -85,B 0,C 180,E1 -19227.447,E2 -19227.447} C_VEL
LIN {X 0,Y 283.566,Z 481.37,A -85,B 0,C 180,E1 -19229.465,E2 -19229.465} C_VEL
LIN {X 0,Y 276.471,Z 491.052,A -85,B 0,C 180,E1 -19231.948,E2 -19231.948} C_VEL
LIN {X 0,Y 270.128,Z 499.128,A -85,B 0,C 180,E1 -19234.578,E2 -19234.578} C_VEL
LIN {X 0,Y 264.462,Z 505.773,A -85,B 0,C 180,E1 -19237.336,E2 -19237.336} C_VEL
LIN {X 0,Y 259.529,Z 511.056,A -85,B 0,C 180,E1 -19240.215,E2 -19240.215} C_VEL
LIN {X 0,Y 256.231,Z 514.172,A -85,B 0,C 180,E1 -19242.44,E2 -19242.44} C_VEL
LIN {X 0,Y 252.384,Z 517.13,A -85,B 0,C 180,E1 -19245.487,E2 -19245.487} C_VEL
LIN {X 0,Y 249.329,Z 518.719,A -85,B 0,C 180,E1 -19248.621,E2 -19248.621} C_VEL
LIN {X 0,Y 247.017,Z 518.94,A -85,B 0,C 180,E1 -19251.822,E2 -19251.822} C_VEL
LIN {X 0,Y 245.257,Z 517.751,A -85,B 0,C 180,E1 -19255.069,E2 -19255.069} C_VEL
LIN {X 0,Y 244.422,Z 516.628,A -85,B 0,C 180,E1 -19256.704,E2 -19256.704} C_VEL
LIN {X 0,Y 243.473,Z 513.138,A -85,B 0,C 180,E1 -19260.001,E2 -19260.001} C_VEL
LIN {X 0,Y 243.141,Z 509.495,A -85,B 0,C 180,E1 -19262.486,E2 -19262.486} C_VEL
LIN {X 0,Y 243.133,Z 504.879,A -85,B 0,C 180,E1 -19264.975,E2 -19264.975} C_VEL
LIN {X 0,Y 243.212,Z 498.214,A -85,B 0,C 180,E1 -19267.89,E2 -19267.89} C_VEL
LIN {X 0,Y 244.067,Z 489.929,A -85,B 0,C 180,E1 -19270.788,E2 -19270.788} C_VEL
LIN {X 0,Y 245.007,Z 479.899,A -85,B 0,C 180,E1 -19273.69,E2 -19273.69} C_VEL
LIN {X 0,Y 246.223,Z 469.551,A -85,B 0,C 180,E1 -19276.159,E2 -19276.159} C_VEL
LIN {X 0,Y 247.65,Z 457.176,A -85,B 0,C 180,E1 -19278.619,E2 -19278.619} C_VEL
LIN {X 0,Y 249.292,Z 445.01,A -85,B 0,C 180,E1 -19280.635,E2 -19280.635} C_VEL
LIN {X 0,Y 250.904,Z 430.457,A -85,B 0,C 180,E1 -19282.641,E2 -19282.641} C_VEL
LIN {X 0,Y 252.16,Z 418.133,A -85,B 0,C 180,E1 -19284.056,E2 -19284.056} C_VEL
LIN {X 0,Y 249.308,Z 403.143,A -85,B 0,C 180,E1 -19285.794,E2 -19285.794} C_VEL
LIN {X 0,Y 245.529,Z 386.497,A -85,B 0,C 180,E1 -19287.453,E2 -19287.453} C_VEL
LIN {X 0,Y 243.389,Z 377.512,A -85,B 0,C 180,E1 -19288.238,E2 -19288.238} C_VEL
LIN {X 0,Y 243.934,Z 372.056,A -85,B 0,C 180,E1 -19292.209,E2 -19292.209} C_VEL
LIN {X 0,Y 244.364,Z 368.2,A -85,B 0,C 180,E1 -19295.115,E2 -19295.115} C_VEL
LIN {X 0,Y 244.359,Z 364.114,A -85,B 0,C 180,E1 -19298.357,E2 -19298.357} C_VEL
LIN {X 0,Y 246.252,Z 367.743,A -85,B 0,C 180,E1 -19301.028,E2 -19301.028} C_VEL
LIN {X 0,Y 247.815,Z 372.177,A -85,B 0,C 180,E1 -19303.924,E2 -19303.924} C_VEL
LIN {X 0,Y 249.175,Z 379.565,A -85,B 0,C 180,E1 -19308.368,E2 -19308.368} C_VEL
LIN {X 0,Y 250.042,Z 385.89,A -85,B 0,C 180,E1 -19311.907,E2 -19311.907} C_VEL
LIN {X 0,Y 249.726,Z 393.521,A -85,B 0,C 180,E1 -19315.743,E2 -19315.743} C_VEL
LIN {X 0,Y 249.474,Z 403.149,A -85,B 0,C 180,E1 -19320.281,E2 -19320.281} C_VEL
LIN {X 0,Y 254.541,Z 415.925,A -85,B 0,C 180,E1 -19321.532,E2 -19321.532} C_VEL
LIN {X 0,Y 257.875,Z 427.015,A -85,B 0,C 180,E1 -19322.769,E2 -19322.769} C_VEL
LIN {X 0,Y 258.889,Z 431.048,A -85,B 0,C 180,E1 -19323.263,E2 -19323.263} C_VEL
LIN {X 0,Y 257.542,Z 443.44,A -85,B 0,C 180,E1 -19324.487,E2 -19324.487} C_VEL
LIN {X 0,Y 255.946,Z 454.387,A -85,B 0,C 180,E1 -19325.889,E2 -19325.889} C_VEL
LIN {X 0,Y 254.046,Z 465.148,A -85,B 0,C 180,E1 -19327.639,E2 -19327.639} C_VEL
LIN {X 0,Y 252.62,Z 472.939,A -85,B 0,C 180,E1 -19329.221,E2 -19329.221} C_VEL
LIN {X 0,Y 250.701,Z 481.065,A -85,B 0,C 180,E1 -19331.189,E2 -19331.189} C_VEL
LIN {X 0,Y 248.755,Z 488.96,A -85,B 0,C 180,E1 -19333.585,E2 -19333.585} C_VEL
LIN {X 0,Y 247.249,Z 495.272,A -85,B 0,C 180,E1 -19336.015,E2 -19336.015} C_VEL
LIN {X 0,Y 245.665,Z 500.335,A -85,B 0,C 180,E1 -19338.444,E2 -19338.444} C_VEL
LIN {X 0,Y 244.487,Z 504.236,A -85,B 0,C 180,E1 -19340.899,E2 -19340.899} C_VEL
LIN {X 0,Y 243.861,Z 507.068,A -85,B 0,C 180,E1 -19343.376,E2 -19343.376} C_VEL
LIN {X 0,Y 243.453,Z 508.456,A -85,B 0,C 180,E1 -19345.028,E2 -19345.028} C_VEL
LIN {X 0,Y 243.069,Z 510.015,A -85,B 0,C 180,E1 -19348.339,E2 -19348.339} C_VEL
LIN {X 0,Y 243.01,Z 510.243,A -85,B 0,C 180,E1 -19349.996,E2 -19349.996} C_VEL
LIN {X 0,Y 243.169,Z 509.486,A -85,B 0,C 180,E1 -19353.31,E2 -19353.31} C_VEL
LIN {X 0,Y 243.858,Z 507.199,A -85,B 0,C 180,E1 -19356.616,E2 -19356.616} C_VEL
LIN {X 0,Y 244.464,Z 504.417,A -85,B 0,C 180,E1 -19359.093,E2 -19359.093} C_VEL
LIN {X 0,Y 245.643,Z 500.576,A -85,B 0,C 180,E1 -19361.549,E2 -19361.549} C_VEL
LIN {X 0,Y 247.197,Z 495.578,A -85,B 0,C 180,E1 -19363.98,E2 -19363.98} C_VEL
LIN {X 0,Y 248.715,Z 489.326,A -85,B 0,C 180,E1 -19366.409,E2 -19366.409} C_VEL
LIN {X 0,Y 250.637,Z 481.516,A -85,B 0,C 180,E1 -19368.808,E2 -19368.808} C_VEL
LIN {X 0,Y 252.463,Z 473.511,A -85,B 0,C 180,E1 -19370.785,E2 -19370.785} C_VEL
LIN {X 0,Y 254.177,Z 464.765,A -85,B 0,C 180,E1 -19372.555,E2 -19372.555} C_VEL
LIN {X 0,Y 255.999,Z 453.892,A -85,B 0,C 180,E1 -19374.313,E2 -19374.313} C_VEL
LIN {X 0,Y 257.651,Z 443.078,A -85,B 0,C 180,E1 -19375.675,E2 -19375.675} C_VEL
LIN {X 0,Y 258.829,Z 432.743,A -85,B 0,C 180,E1 -19376.702,E2 -19376.702} C_VEL
LIN {X 0,Y 258.875,Z 430.761,A -85,B 0,C 180,E1 -19376.892,E2 -19376.892} C_VEL
LIN {X 0,Y 255.437,Z 418.664,A -85,B 0,C 180,E1 -19378.304,E2 -19378.304} C_VEL
LIN {X 0,Y 250.909,Z 406.55,A -85,B 0,C 180,E1 -19379.538,E2 -19379.538} C_VEL
LIN {X 0,Y 249.538,Z 403.079,A -85,B 0,C 180,E1 -19379.89,E2 -19379.89} C_VEL
LIN {X 0,Y 249.726,Z 393.867,A -85,B 0,C 180,E1 -19384.248,E2 -19384.248} C_VEL
LIN {X 0,Y 250.015,Z 386.211,A -85,B 0,C 180,E1 -19388.085,E2 -19388.085} C_VEL
LIN {X 0,Y 249.542,Z 381.862,A -85,B 0,C 180,E1 -19390.498,E2 -19390.498} C_VEL
LIN {X 0,Y 248.563,Z 376.087,A -85,B 0,C 180,E1 -19393.862,E2 -19393.862} C_VEL
LIN {X 0,Y 247.319,Z 369.785,A -85,B 0,C 180,E1 -19397.625,E2 -19397.625} C_VEL
LIN {X 0,Y 246.04,Z 364.351,A -85,B 0,C 180,E1 -19401.066,E2 -19401.066} C_VEL
LIN {X 0,Y 244.534,Z 358.599,A -85,B 0,C 180,E1 -19404.913,E2 -19404.913} C_VEL
LIN {X 0,Y 243.22,Z 354.752,A -85,B 0,C 180,E1 -19407.533,E2 -19407.533} C_VEL
LIN {X 0,Y 242.013,Z 350.643,A -85,B 0,C 180,E1 -19410.417,E2 -19410.417} C_VEL
LIN {X 0,Y 242.05,Z 350.638,A -85,B 0,C 180,E1 -19414.18,E2 -19414.18} C_VEL
LIN {X 0,Y 242.071,Z 350.637,A -85,B 0,C 180,E1 -19418.273,E2 -19418.273} C_VEL
LIN {X 0,Y 242.144,Z 350.636,A -85,B 0,C 180,E1 -19423.276,E2 -19423.276} C_VEL
LIN {X 0,Y 242.166,Z 350.634,A -85,B 0,C 180,E1 -19428.278,E2 -19428.278} C_VEL
LIN {X 0,Y 242.406,Z 350.591,A -85,B 0,C 180,E1 -19431.664,E2 -19431.664} C_VEL
LIN {X 0,Y 242.235,Z 350.607,A -85,B 0,C 180,E1 -19435.006,E2 -19435.006} C_VEL
LIN {X 0,Y 242.613,Z 350.578,A -85,B 0,C 180,E1 -19438.339,E2 -19438.339} C_VEL
LIN {X 0,Y 242.626,Z 350.56,A -85,B 0,C 180,E1 -19441.659,E2 -19441.659} C_VEL
LIN {X 0,Y 242.414,Z 350.599,A -85,B 0,C 180,E1 -19446.659,E2 -19446.659} C_VEL
LIN {X 0,Y 242.292,Z 350.619,A -85,B 0,C 180,E1 -19450.022,E2 -19450.022} C_VEL
LIN {X 0,Y 242.177,Z 350.747,A -85,B 0,C 180,E1 -19454.924,E2 -19454.924} C_VEL
LIN {X 0,Y 243.671,Z 356.803,A -85,B 0,C 180,E1 -19459.37,E2 -19459.37} C_VEL
LIN {X 0,Y 245.331,Z 363.163,A -85,B 0,C 180,E1 -19463.644,E2 -19463.644} C_VEL
LIN {X 0,Y 246.765,Z 368.742,A -85,B 0,C 180,E1 -19467.109,E2 -19467.109} C_VEL
LIN {X 0,Y 247.516,Z 371.437,A -85,B 0,C 180,E1 -19468.717,E2 -19468.717} C_VEL
LIN {X 0,Y 247.512,Z 373.82,A -85,B 0,C 180,E1 -19469.967,E2 -19469.967} C_VEL
LIN {X 0,Y 245.776,Z 378.317,A -85,B 0,C 180,E1 -19471.979,E2 -19471.979} C_VEL
LIN {X 0,Y 244.228,Z 382.047,A -85,B 0,C 180,E1 -19473.6,E2 -19473.6} C_VEL
LIN {X 0,Y 243.818,Z 384.705,A -85,B 0,C 180,E1 -19474.851,E2 -19474.851} C_VEL
LIN {X 0,Y 243.935,Z 385.536,A -85,B 0,C 180,E1 -19475.274,E2 -19475.274} C_VEL
LIN {X 0,Y 246.225,Z 394.122,A -85,B 0,C 180,E1 -19479.595,E2 -19479.595} C_VEL
LIN {X 0,Y 248.709,Z 403.179,A -85,B 0,C 180,E1 -19483.813,E2 -19483.813} C_VEL
LIN {X 0,Y 250.525,Z 409.635,A -85,B 0,C 180,E1 -19486.579,E2 -19486.579} C_VEL
LIN {X 0,Y 252.455,Z 415.2,A -85,B 0,C 180,E1 -19487.068,E2 -19487.068} C_VEL
LIN {X 0,Y 253.996,Z 432.906,A -85,B 0,C 180,E1 -19488.231,E2 -19488.231} C_VEL
LIN {X 0,Y 255.353,Z 449.732,A -85,B 0,C 180,E1 -19489.642,E2 -19489.642} C_VEL
LIN {X 0,Y 256.619,Z 465.692,A -85,B 0,C 180,E1 -19491.278,E2 -19491.278} C_VEL
